(* Logix 5000 project; controller cal1615 1756-L62 rev 20.19; software revision 20.05; part 8 of 81 *)
(* tags used below, declared in another part *)
   AFI : BOOL;   // Always False Bit
   AutoT : PIDE_AUTOTUNE;
   FAULT : BOOL;   // Fault AFI
   HMI : BOOL;   // AFI HMI
   p01_dint_to_hmi : DINT[16];   // System Dint to HMI
   p01_param_heater_hl : REAL;   // Machine Parameter Heater HighTemperature Max Limit
   p01_param_process_air_hl : REAL;   // Machine Parameter Process Air High Limit
   p01_param_process_air_max : REAL;   // Machine Parameter Process Air High Temperature Max Setpoint Limit
   p01_param_temp_limit : REAL;   // Machine Parameter Maximum Temperature for Fan Operation
   p01_recipe_active : recipe;   // Active Recipe
   p01r01 : routine;
   p01r02 : routine;   // System Misc Control
   p01r02_all_fans_stopped : BOOL;   // System Misc Control All Fans Stopped
   p01r02_batch_run_time : DINT;   // System Misc Control Batch Minutes
   p01r02_batch_run_time_hrs : DINT;   // System Misc Control Batch Hours
   p01r02_ethernet_comm : DINT;
   p01r02_fault_exists : BOOL;
   p01r02_flash_bit : BOOL;   // System Misc Control Flash Bit
   p01r02_flash_timer_off : TIMER;   // System Misc Control Flash Timer Off
   p01r02_flash_timer_on : TIMER;   // System Misc Control Flash Timer On
   p01r02_plc_faults : DINT;   // System Misc Control PLC Faults
   p01r02_plc_scan_time : DINT;   // System PLC Scan Time
   p01r02_plc_scan_time_in_sec : REAL;   // System PLC Scan Time in Seconds
   p01r02_timer_batch : TIMER;   // System Misc Control Batch Timer Seconds
   p01r02_timer_fault : TIMER[25];   // System Misc Control Fault Dwell Timer
   p01r02_timer_half_second_off : TIMER;   // System Misc Control Timer Second Pulse Off
   p01r02_timer_half_second_on : TIMER;   // System Misc Control Timer 1/2 Second Pulse On
   p01r02_timer_second : TIMER[2];   // System Misc Control Timer Second Pulse
   p01r02_unack_fault : BOOL;   // System Misc Control Unacknowledged Fault Exists
   p01r02_unack_warning : BOOL;   // System Misc Control Unacknowledged Warning Exists
   p01r02_vfd_comm_2 : DINT[50];
   p01r02_warnings_exists : BOOL;
   p01r03 : routine;   // System Inputs
   p01r04 : routine;   // System Outputs
   p01r05 : routine;   // System Dint to HMI
   p01r06 : routine;   // System Real to HMI
   p01r07 : routine;   // System Alarms
   p01r08 : routine;   // System Warnings
   p01r09 : routine;   // System Modes
   p01r09_pb_global_reset : BOOL;   // System Modes PB: Global Fault Reset
   p01r10 : routine;   // System Annunciators
   p01r11 : routine;   // System Timer Presets
   p01r12 : routine;   // System Line Accel Decel Control
   p01r13 : routine;   // System Line Start Sequence
   p01r13_line_running : BOOL;   // System Line Start Sequence Line Running
   p02_dint_from_hmi : hmi_dint;
   p11r31_request_auto_run : BOOL;   // Zone 1 Exhaust Fan Run Request
   p11r32_request_auto_run : BOOL;   // Zone 1 Recirc Fan Run Request
   p12r31_request_auto_run : BOOL;   // Zone 2 Exhaust Fan Run Request
   p12r32_request_auto_run : BOOL;   // Zone 2 Recirc Fan Run Request
   p13r31_request_auto_run : BOOL;   // Zone 3 Exhaust Fan Run Request
   p13r32_request_auto_run : BOOL;   // Zone 3 Recirc Fan Run Request
   p23_do_enable_impreg_exhaust_fan : BOOL;   // Impreg Enclosure Digital Output Exhaust Fan Enable
   p23r13_request_auto_run : BOOL;   // Impreg Supply Fan VFD Request Auto Run
   p25_ai_ts2_lc : REAL;   // System Metering Roll VFD Minimum Start Tension
   p25r10_pid_manual_request : BOOL;
   p25r10_tension_request : BOOL;
   p25r20_pide_cv : REAL;

   p29r16_torque_acc_rate : REAL := 0.05;
   p29r16_torque_boost_acc_rate : REAL := 5000.0;
   p29r16_torque_boost_dec_rate : REAL := 2.0;
   p29r16_torque_boost_ref : REAL := 90.0;   // Winder Winder A VFD Request Jog REV
   p29r16_torque_boost_timer : TIMER := (PRE := 500);   // Zone 1 Exhaust VFD PB: Auto Stop
   p29r16_torque_dec_rate : REAL := 0.05;
   p29r16_torque_fast_acc_rate : REAL := 0.8;
   p29r16_torque_fast_dec_rate : REAL := 1.6;
   p29r16_torque_high_ref : REAL := 100.0;
   p29r16_torque_low_ref : REAL := 1.0;
   p29r16_torque_mode_acc_rate : REAL := 5000.0;
   p29r16_torque_mode_dec_rate : REAL := 4.0;
   p29r16_torque_ramp : SYS_ACC_DEC_RAMP := (IN_selected_line_speed := 100.0, IN_param_master_accel_rate := 0.05, IN_param_master_decel_rate := 0.05, IN_last_scan_s := 0.03255);
   p29r16_torque_soak_acc_rate : REAL := 0.05;
   p29r16_torque_soak_dec_rate : REAL := 0.05;
   p29r16_torque_start_timer : TIMER := (PRE := 200);   // Timer Winder B Torque Start Timer
   p29r16_vfd_start_request : BOOL := 1;
   p29r16_wdrb_accel_decel : SYS_ACC_DEC_RAMP := (IN_selected_line_speed := 16.283354, IN_param_master_accel_rate := 25.0, IN_param_master_decel_rate := 25.0, IN_last_scan_s := 0.03455);   // Winder Winder B VFD Accel Decel Ramp
   p29r16_wdrb_active : BOOL := 1;   // Winder Winder B VFD Active
   p29r16_wdrb_ramped_speed : REAL := 15.371705;   // Winder Winder B VFD Ramped Speed
   p29r16_zero_speed : BOOL;   // Winder Winder A VFD At Zero BSpeed
   p29r17 : routine := (comment := -1073741777);   // Winder Winder A Diameter
        .FAULT   // Winder Winder Turret VFD
        .UNACK_FAULT   // Winder Winder A Diameter Unacknowleged Faults Exist
        .UNACK_WARNING   // Winder Winder A Diameter Unacknowleged Warnings Exist
   p29r17_ave_control : CONTROL := (LEN := 19);   // Winder Winder A Diameter Calculation AVE Control
   p29r17_diameter_clac_active : BOOL;   // Winder Winder A Diameter Calculation Calc Active
   p29r17_selected_core_diameter : REAL := 3.25;   // Winder Winder A Diameter Calculation Selected Core Diameter
   p29r17_stack_ctrl : CONTROL := (LEN := 20, POS := 19);   // Winder Winder A Diameter Calculation Stack Control
   p29r17_timer : TIMER[5] := ([0].PRE := 20000, [1].PRE := 500);   // Winder Winder A Diameter Calculation Timers
        [1]   // Winder Winder A Diameter Calculation Sample Timer
   p29r17_timer_fault : TIMER[4];   // Winder Winder A Diameter Calculation Fault Dwell Timer
   p29r17_timer_warning : TIMER[4];   // Winder Winder A Diameter Calculation Warning Dwell Timer
   p29r17_web_speed_at_winder : REAL;   // Winder Winder A Diameter True Web Speed at the Winder Line Speed plus Accumulator Payout [fpm]
   p29r17_winder_a_actual_diam_inch : REAL := 6.327387;   // Winder Winder A Diameter Calculation Actual Diameter [in]
   p29r17_winder_a_avg_diam_inch : REAL := 6.2460294;   // Winder Winder A Diameter Calculation Winder A Average Diameter [in]
   p29r17_winder_a_calc_diam_inch : REAL := 6.327387;   // Winder Winder A Diameter Calculated Diameter Inch
   p29r17_winder_a_diam_avg_stack : REAL[1000] := ([0] := 6.227294, [1] := 6.2310367, [2] := 6.224801, [3] := 6.228541, [4] := 6.246055, [5] := 6.25359, [6] := 6.2360344, [7] := 6.2185774, [8] := 6.2148495, [9] := 6.216091, [10] := 6.247309, [11] := 6.2448, [12] := 6.2335353, [13] := 6.247309, [14] := 6.2737756, [15] := 6.277575, [16] := 6.304299, [17] := 6.3441668, [18] := 6.323527, [20] := 3.25, [21] := 3.25, [22] := 3.25, [23] := 3.25, [24] := 3.25, [25] := 3.25, [26] := 3.25, [27] := 3.25, [28] := 3.25, [29] := 3.25, [30] := 3.25, [31] := 3.25, [32] := 3.25, [33] := 3.25, [34] := 3.25, [35] := 3.25, [36] := 3.25, [37] := 3.25, [38] := 3.25, [39] := 3.25, [40] := 3.25, [41] := 3.25, [42] := 3.25, [43] := 3.25, [44] := 3.25, [45] := 3.25, [46] := 3.25, [47] := 3.25, [48] := 3.25, [49] := 3.25, [50] := 3.25, [51] := 3.25, [52] := 3.25, [53] := 3.25, [54] := 3.25, [55] := 3.25, [56] := 3.25, [57] := 3.25, [58] := 3.25, [59] := 3.25, [60] := 3.25,
        [61] := 3.25, [62] := 3.25, [63] := 3.25, [64] := 3.25, [65] := 3.25, [66] := 3.25, [67] := 3.25, [68] := 3.25, [69] := 3.25, [70] := 3.25, [71] := 3.25, [72] := 3.25, [73] := 3.25, [74] := 3.25, [75] := 3.25, [76] := 3.25, [77] := 3.25, [78] := 3.25, [79] := 3.25, [80] := 3.25, [81] := 3.25, [82] := 3.25, [83] := 3.25, [84] := 3.25, [85] := 3.25, [86] := 3.25, [87] := 3.25, [88] := 3.25, [89] := 3.25, [90] := 3.25, [91] := 3.25, [92] := 3.25, [93] := 3.25, [94] := 3.25, [95] := 3.25, [96] := 3.25, [97] := 3.25, [98] := 3.25, [99] := 3.25, [100] := 3.25, [101] := 3.25, [102] := 3.25, [103] := 3.25, [104] := 3.25, [105] := 3.25, [106] := 3.25, [107] := 3.25, [108] := 3.25, [109] := 3.25, [110] := 3.25, [111] := 3.25, [112] := 3.25, [113] := 3.25, [114] := 3.25, [115] := 3.25, [116] := 3.25, [117] := 3.25, [118] := 3.25, [119] := 3.25, [120] := 3.25,
        [121] := 3.25, [122] := 3.25, [123] := 3.25, [124] := 3.25, [125] := 3.25, [126] := 3.25, [127] := 3.25, [128] := 3.25, [129] := 3.25, [130] := 3.25, [131] := 3.25, [132] := 3.25, [133] := 3.25, [134] := 3.25, [135] := 3.25, [136] := 3.25, [137] := 3.25, [138] := 3.25, [139] := 3.25, [140] := 3.25, [141] := 3.25, [142] := 3.25, [143] := 3.25, [144] := 3.25, [145] := 3.25, [146] := 3.25, [147] := 3.25, [148] := 3.25, [149] := 3.25, [150] := 3.25, [151] := 3.25, [152] := 3.25, [153] := 3.25, [154] := 3.25, [155] := 3.25, [156] := 3.25, [157] := 3.25, [158] := 3.25, [159] := 3.25, [160] := 3.25, [161] := 3.25, [162] := 3.25, [163] := 3.25, [164] := 3.25, [165] := 3.25, [166] := 3.25, [167] := 3.25, [168] := 3.25, [169] := 3.25, [170] := 3.25, [171] := 3.25, [172] := 3.25, [173] := 3.25, [174] := 3.25, [175] := 3.25, [176] := 3.25, [177] := 3.25, [178] := 3.25, [179] := 3.25, [180] := 3.25,
        [181] := 3.25, [182] := 3.25, [183] := 3.25, [184] := 3.25, [185] := 3.25, [186] := 3.25, [187] := 3.25, [188] := 3.25, [189] := 3.25, [190] := 3.25, [191] := 3.25, [192] := 3.25, [193] := 3.25, [194] := 3.25, [195] := 3.25, [196] := 3.25, [197] := 3.25, [198] := 3.25, [199] := 3.25, [200] := 3.25, [201] := 3.25, [202] := 3.25, [203] := 3.25, [204] := 3.25, [205] := 3.25, [206] := 3.25, [207] := 3.25, [208] := 3.25, [209] := 3.25, [210] := 3.25, [211] := 3.25, [212] := 3.25, [213] := 3.25, [214] := 3.25, [215] := 3.25, [216] := 3.25, [217] := 3.25, [218] := 3.25, [219] := 3.25, [220] := 3.25, [221] := 3.25, [222] := 3.25, [223] := 3.25, [224] := 3.25, [225] := 3.25, [226] := 3.25, [227] := 3.25, [228] := 3.25, [229] := 3.25, [230] := 3.25, [231] := 3.25, [232] := 3.25, [233] := 3.25, [234] := 3.25, [235] := 3.25, [236] := 3.25, [237] := 3.25, [238] := 3.25, [239] := 3.25, [240] := 3.25,
        [241] := 3.25, [242] := 3.25, [243] := 3.25, [244] := 3.25, [245] := 3.25, [246] := 3.25, [247] := 3.25, [248] := 3.25, [249] := 3.25, [250] := 3.25, [251] := 3.25, [252] := 3.25, [253] := 3.25, [254] := 3.25, [255] := 3.25, [256] := 3.25, [257] := 3.25, [258] := 3.25, [259] := 3.25, [260] := 3.25, [261] := 3.25, [262] := 3.25, [263] := 3.25, [264] := 3.25, [265] := 3.25, [266] := 3.25, [267] := 3.25, [268] := 3.25, [269] := 3.25, [270] := 3.25, [271] := 3.25, [272] := 3.25, [273] := 3.25, [274] := 3.25, [275] := 3.25, [276] := 3.25, [277] := 3.25, [278] := 3.25, [279] := 3.25, [280] := 3.25, [281] := 3.25, [282] := 3.25, [283] := 3.25, [284] := 3.25, [285] := 3.25, [286] := 3.25, [287] := 3.25, [288] := 3.25, [289] := 3.25, [290] := 3.25, [291] := 3.25, [292] := 3.25, [293] := 3.25, [294] := 3.25, [295] := 3.25, [296] := 3.25, [297] := 3.25, [298] := 3.25, [299] := 3.25, [300] := 3.25,
        [301] := 3.25, [302] := 3.25, [303] := 3.25, [304] := 3.25, [305] := 3.25, [306] := 3.25, [307] := 3.25, [308] := 3.25, [309] := 3.25, [310] := 3.25, [311] := 3.25, [312] := 3.25, [313] := 3.25, [314] := 3.25, [315] := 3.25, [316] := 3.25, [317] := 3.25, [318] := 3.25, [319] := 3.25, [320] := 3.25, [321] := 3.25, [322] := 3.25, [323] := 3.25, [324] := 3.25, [325] := 3.25, [326] := 3.25, [327] := 3.25, [328] := 3.25, [329] := 3.25, [330] := 3.25, [331] := 3.25, [332] := 3.25, [333] := 3.25, [334] := 3.25, [335] := 3.25, [336] := 3.25, [337] := 3.25, [338] := 3.25, [339] := 3.25, [340] := 3.25, [341] := 3.25, [342] := 3.25, [343] := 3.25, [344] := 3.25, [345] := 3.25, [346] := 3.25, [347] := 3.25, [348] := 3.25, [349] := 3.25, [350] := 3.25, [351] := 3.25, [352] := 3.25, [353] := 3.25, [354] := 3.25, [355] := 3.25, [356] := 3.25, [357] := 3.25, [358] := 3.25, [359] := 3.25, [360] := 3.25,
        [361] := 3.25, [362] := 3.25, [363] := 3.25, [364] := 3.25, [365] := 3.25, [366] := 3.25, [367] := 3.25, [368] := 3.25, [369] := 3.25, [370] := 3.25, [371] := 3.25, [372] := 3.25, [373] := 3.25, [374] := 3.25, [375] := 3.25, [376] := 3.25, [377] := 3.25, [378] := 3.25, [379] := 3.25, [380] := 3.25, [381] := 3.25, [382] := 3.25, [383] := 3.25, [384] := 3.25, [385] := 3.25, [386] := 3.25, [387] := 3.25, [388] := 3.25, [389] := 3.25, [390] := 3.25, [391] := 3.25, [392] := 3.25, [393] := 3.25, [394] := 3.25, [395] := 3.25, [396] := 3.25, [397] := 3.25, [398] := 3.25, [399] := 3.25, [400] := 3.25, [401] := 3.25, [402] := 3.25, [403] := 3.25, [404] := 3.25, [405] := 3.25, [406] := 3.25, [407] := 3.25, [408] := 3.25, [409] := 3.25, [410] := 3.25, [411] := 3.25, [412] := 3.25, [413] := 3.25, [414] := 3.25, [415] := 3.25, [416] := 3.25, [417] := 3.25, [418] := 3.25, [419] := 3.25, [420] := 3.25,
        [421] := 3.25, [422] := 3.25, [423] := 3.25, [424] := 3.25, [425] := 3.25, [426] := 3.25, [427] := 3.25, [428] := 3.25, [429] := 3.25, [430] := 3.25, [431] := 3.25, [432] := 3.25, [433] := 3.25, [434] := 3.25, [435] := 3.25, [436] := 3.25, [437] := 3.25, [438] := 3.25, [439] := 3.25, [440] := 3.25, [441] := 3.25, [442] := 3.25, [443] := 3.25, [444] := 3.25, [445] := 3.25, [446] := 3.25, [447] := 3.25, [448] := 3.25, [449] := 3.25, [450] := 3.25, [451] := 3.25, [452] := 3.25, [453] := 3.25, [454] := 3.25, [455] := 3.25, [456] := 3.25, [457] := 3.25, [458] := 3.25, [459] := 3.25, [460] := 3.25, [461] := 3.25, [462] := 3.25, [463] := 3.25, [464] := 3.25, [465] := 3.25, [466] := 3.25, [467] := 3.25, [468] := 3.25, [469] := 3.25, [470] := 3.25, [471] := 3.25, [472] := 3.25, [473] := 3.25, [474] := 3.25, [475] := 3.25, [476] := 3.25, [477] := 3.25, [478] := 3.25, [479] := 3.25, [480] := 3.25,
        [481] := 3.25, [482] := 3.25, [483] := 3.25, [484] := 3.25, [485] := 3.25, [486] := 3.25, [487] := 3.25, [488] := 3.25, [489] := 3.25, [490] := 3.25, [491] := 3.25, [492] := 3.25, [493] := 3.25, [494] := 3.25, [495] := 3.25, [496] := 3.25, [497] := 3.25, [498] := 3.25, [499] := 3.25, [500] := 3.25, [501] := 3.25, [502] := 3.25, [503] := 3.25, [504] := 3.25, [505] := 3.25, [506] := 3.25, [507] := 3.25, [508] := 3.25, [509] := 3.25, [510] := 3.25, [511] := 3.25, [512] := 3.25, [513] := 3.25, [514] := 3.25, [515] := 3.25, [516] := 3.25, [517] := 3.25, [518] := 3.25, [519] := 3.25, [520] := 3.25, [521] := 3.25, [522] := 3.25, [523] := 3.25, [524] := 3.25, [525] := 3.25, [526] := 3.25, [527] := 3.25, [528] := 3.25, [529] := 3.25, [530] := 3.25, [531] := 3.25, [532] := 3.25, [533] := 3.25, [534] := 3.25, [535] := 3.25, [536] := 3.25, [537] := 3.25, [538] := 3.25, [539] := 3.25, [540] := 3.25,
        [541] := 3.25, [542] := 3.25, [543] := 3.25, [544] := 3.25, [545] := 3.25, [546] := 3.25, [547] := 3.25, [548] := 3.25, [549] := 3.25, [550] := 3.25, [551] := 3.25, [552] := 3.25, [553] := 3.25, [554] := 3.25, [555] := 3.25, [556] := 3.25, [557] := 3.25, [558] := 3.25, [559] := 3.25, [560] := 3.25, [561] := 3.25, [562] := 3.25, [563] := 3.25, [564] := 3.25, [565] := 3.25, [566] := 3.25, [567] := 3.25, [568] := 3.25, [569] := 3.25, [570] := 3.25, [571] := 3.25, [572] := 3.25, [573] := 3.25, [574] := 3.25, [575] := 3.25, [576] := 3.25, [577] := 3.25, [578] := 3.25, [579] := 3.25, [580] := 3.25, [581] := 3.25, [582] := 3.25, [583] := 3.25, [584] := 3.25, [585] := 3.25, [586] := 3.25, [587] := 3.25, [588] := 3.25, [589] := 3.25, [590] := 3.25, [591] := 3.25, [592] := 3.25, [593] := 3.25, [594] := 3.25, [595] := 3.25, [596] := 3.25, [597] := 3.25, [598] := 3.25, [599] := 3.25, [600] := 3.25,
        [601] := 3.25, [602] := 3.25, [603] := 3.25, [604] := 3.25, [605] := 3.25, [606] := 3.25, [607] := 3.25, [608] := 3.25, [609] := 3.25, [610] := 3.25, [611] := 3.25, [612] := 3.25, [613] := 3.25, [614] := 3.25, [615] := 3.25, [616] := 3.25, [617] := 3.25, [618] := 3.25, [619] := 3.25, [620] := 3.25, [621] := 3.25, [622] := 3.25, [623] := 3.25, [624] := 3.25, [625] := 3.25, [626] := 3.25, [627] := 3.25, [628] := 3.25, [629] := 3.25, [630] := 3.25, [631] := 3.25, [632] := 3.25, [633] := 3.25, [634] := 3.25, [635] := 3.25, [636] := 3.25, [637] := 3.25, [638] := 3.25, [639] := 3.25, [640] := 3.25, [641] := 3.25, [642] := 3.25, [643] := 3.25, [644] := 3.25, [645] := 3.25, [646] := 3.25, [647] := 3.25, [648] := 3.25, [649] := 3.25, [650] := 3.25, [651] := 3.25, [652] := 3.25, [653] := 3.25, [654] := 3.25, [655] := 3.25, [656] := 3.25, [657] := 3.25, [658] := 3.25, [659] := 3.25, [660] := 3.25,
        [661] := 3.25, [662] := 3.25, [663] := 3.25, [664] := 3.25, [665] := 3.25, [666] := 3.25, [667] := 3.25, [668] := 3.25, [669] := 3.25, [670] := 3.25, [671] := 3.25, [672] := 3.25, [673] := 3.25, [674] := 3.25, [675] := 3.25, [676] := 3.25, [677] := 3.25, [678] := 3.25, [679] := 3.25, [680] := 3.25, [681] := 3.25, [682] := 3.25, [683] := 3.25, [684] := 3.25, [685] := 3.25, [686] := 3.25, [687] := 3.25, [688] := 3.25, [689] := 3.25, [690] := 3.25, [691] := 3.25, [692] := 3.25, [693] := 3.25, [694] := 3.25, [695] := 3.25, [696] := 3.25, [697] := 3.25, [698] := 3.25, [699] := 3.25, [700] := 3.25, [701] := 3.25, [702] := 3.25, [703] := 3.25, [704] := 3.25, [705] := 3.25, [706] := 3.25, [707] := 3.25, [708] := 3.25, [709] := 3.25, [710] := 3.25, [711] := 3.25, [712] := 3.25, [713] := 3.25, [714] := 3.25, [715] := 3.25, [716] := 3.25, [717] := 3.25, [718] := 3.25, [719] := 3.25, [720] := 3.25,
        [721] := 3.25, [722] := 3.25, [723] := 3.25, [724] := 3.25, [725] := 3.25, [726] := 3.25, [727] := 3.25, [728] := 3.25, [729] := 3.25, [730] := 3.25, [731] := 3.25, [732] := 3.25, [733] := 3.25, [734] := 3.25, [735] := 3.25, [736] := 3.25, [737] := 3.25, [738] := 3.25, [739] := 3.25, [740] := 3.25, [741] := 3.25, [742] := 3.25, [743] := 3.25, [744] := 3.25, [745] := 3.25, [746] := 3.25, [747] := 3.25, [748] := 3.25, [749] := 3.25, [750] := 3.25, [751] := 3.25, [752] := 3.25, [753] := 3.25, [754] := 3.25, [755] := 3.25, [756] := 3.25, [757] := 3.25, [758] := 3.25, [759] := 3.25, [760] := 3.25, [761] := 3.25, [762] := 3.25, [763] := 3.25, [764] := 3.25, [765] := 3.25, [766] := 3.25, [767] := 3.25, [768] := 3.25, [769] := 3.25, [770] := 3.25, [771] := 3.25, [772] := 3.25, [773] := 3.25, [774] := 3.25, [775] := 3.25, [776] := 3.25, [777] := 3.25, [778] := 3.25, [779] := 3.25, [780] := 3.25,
        [781] := 3.25, [782] := 3.25, [783] := 3.25, [784] := 3.25, [785] := 3.25, [786] := 3.25, [787] := 3.25, [788] := 3.25, [789] := 3.25, [790] := 3.25, [791] := 3.25, [792] := 3.25, [793] := 3.25, [794] := 3.25, [795] := 3.25, [796] := 3.25, [797] := 3.25, [798] := 3.25, [799] := 3.25, [800] := 3.25, [801] := 3.25, [802] := 3.25, [803] := 3.25, [804] := 3.25, [805] := 3.25, [806] := 3.25, [807] := 3.25, [808] := 3.25, [809] := 3.25, [810] := 3.25, [811] := 3.25, [812] := 3.25, [813] := 3.25, [814] := 3.25, [815] := 3.25, [816] := 3.25, [817] := 3.25, [818] := 3.25, [819] := 3.25, [820] := 3.25, [821] := 3.25, [822] := 3.25, [823] := 3.25, [824] := 3.25, [825] := 3.25, [826] := 3.25, [827] := 3.25, [828] := 3.25, [829] := 3.25, [830] := 3.25, [831] := 3.25, [832] := 3.25, [833] := 3.25, [834] := 3.25, [835] := 3.25, [836] := 3.25, [837] := 3.25, [838] := 3.25, [839] := 3.25, [840] := 3.25,
        [841] := 3.25, [842] := 3.25, [843] := 3.25, [844] := 3.25, [845] := 3.25, [846] := 3.25, [847] := 3.25, [848] := 3.25, [849] := 3.25, [850] := 3.25, [851] := 3.25, [852] := 3.25, [853] := 3.25, [854] := 3.25, [855] := 3.25, [856] := 3.25, [857] := 3.25, [858] := 3.25, [859] := 3.25, [860] := 3.25, [861] := 3.25, [862] := 3.25, [863] := 3.25, [864] := 3.25, [865] := 3.25, [866] := 3.25, [867] := 3.25, [868] := 3.25, [869] := 3.25, [870] := 3.25, [871] := 3.25, [872] := 3.25, [873] := 3.25, [874] := 3.25, [875] := 3.25, [876] := 3.25, [877] := 3.25, [878] := 3.25, [879] := 3.25, [880] := 3.25, [881] := 3.25, [882] := 3.25, [883] := 3.25, [884] := 3.25, [885] := 3.25, [886] := 3.25, [887] := 3.25, [888] := 3.25, [889] := 3.25, [890] := 3.25, [891] := 3.25, [892] := 3.25, [893] := 3.25, [894] := 3.25, [895] := 3.25, [896] := 3.25, [897] := 3.25, [898] := 3.25, [899] := 3.25, [900] := 3.25,
        [901] := 3.25, [902] := 3.25, [903] := 3.25, [904] := 3.25, [905] := 3.25, [906] := 3.25, [907] := 3.25, [908] := 3.25, [909] := 3.25, [910] := 3.25, [911] := 3.25, [912] := 3.25, [913] := 3.25, [914] := 3.25, [915] := 3.25, [916] := 3.25, [917] := 3.25, [918] := 3.25, [919] := 3.25, [920] := 3.25, [921] := 3.25, [922] := 3.25, [923] := 3.25, [924] := 3.25, [925] := 3.25, [926] := 3.25, [927] := 3.25, [928] := 3.25, [929] := 3.25, [930] := 3.25, [931] := 3.25, [932] := 3.25, [933] := 3.25, [934] := 3.25, [935] := 3.25, [936] := 3.25, [937] := 3.25, [938] := 3.25, [939] := 3.25, [940] := 3.25, [941] := 3.25, [942] := 3.25, [943] := 3.25, [944] := 3.25, [945] := 3.25, [946] := 3.25, [947] := 3.25, [948] := 3.25, [949] := 3.25, [950] := 3.25, [951] := 3.25, [952] := 3.25, [953] := 3.25, [954] := 3.25, [955] := 3.25, [956] := 3.25, [957] := 3.25, [958] := 3.25, [959] := 3.25, [960] := 3.25,
        [961] := 3.25, [962] := 3.25, [963] := 3.25, [964] := 3.25, [965] := 3.25, [966] := 3.25, [967] := 3.25, [968] := 3.25, [969] := 3.25, [970] := 3.25, [971] := 3.25, [972] := 3.25, [973] := 3.25, [974] := 3.25, [975] := 3.25, [976] := 3.25, [977] := 3.25, [978] := 3.25, [979] := 3.25, [980] := 3.25, [981] := 3.25, [982] := 3.25, [983] := 3.25, [984] := 3.25, [985] := 3.25, [986] := 3.25, [987] := 3.25, [988] := 3.25, [989] := 3.25, [990] := 3.25, [991] := 3.25, [992] := 3.25, [993] := 3.25, [994] := 3.25, [995] := 3.25, [996] := 3.25, [997] := 3.25, [998] := 3.25, [999] := 3.25);
   p29r17_winder_a_selected_diam_inch : REAL := 3.25;   // Winder Winder A Diameter Calculation Winder Selected Diameter [in]
   p29r17_winder_a_unload : REAL := 6.2049294;
   p29r18 : routine := (comment := -1073741777);   // Winder Winder B Diameter
        .UNACK_FAULT   // Winder Winder B Diameter Unacknowleged Faults Exist
        .UNACK_WARNING   // Winder Winder B Diameter Unacknowleged Warnings Exist
   p29r18_ave_control : CONTROL := (LEN := 19);   // Winder Winder A Diameter Calculation AVE Control
   p29r18_diameter_calc_active : BOOL := 1;   // Winder Winder B Diameter Calculation Calculation Active
   p29r18_min_tension : REAL := 10.0;   // Winder Winder B Diameter Calc Minimum Tension
   p29r18_selected_core_diameter : REAL := 3.25;   // Winder Winder B Diameter Calculation Selected Core Diameter
   p29r18_stack_ctrl : CONTROL := (LEN := 20, POS := 20, EN := 1, DN := 1);   // Winder Winder B Diameter Calculation FiFo Control
   p29r18_timer : TIMER[5] := ([0].PRE := 20000, [0].ACC := 20017, [0].EN := 1, [0].DN := 1, [1].PRE := 500, [1].ACC := 466, [1].EN := 1, [1].TT := 1);   // Winder Winder B Diameter Calculation Timers
   p29r18_timer_fault : TIMER[4];   // Winder Winder B Diameter Calculation Fault Dwell Timer
   p29r18_timer_warning : TIMER[4];   // Winder Winder B Diameter Warning Dwell Timer
   p29r18_web_speed_at_winder : REAL;   // Winder Winder B Diameter True Web Speed at the Winder Line Speed plus Accumulator Payout [fpm]
   p29r18_winder_b_actual_diam_inch : REAL := 7.2323503;   // Winder Winder B Diameter Calculation Actual Diameter [in]
   p29r18_winder_b_avg_diam_inch : REAL := 6.935298;   // Winder Winder B Diameter Calculation Average Diameter [in]
   p29r18_winder_b_calc_diam_inch : REAL := 7.21557;   // Winder Winder B Diameter Calculated Diameter Inch
   p29r18_winder_b_diam_avg_stack : REAL[1000] := ([0] := 7.30026, [1] := 7.30026, [2] := 7.30026, [3] := 7.30026, [4] := 7.30026, [5] := 7.30026, [6] := 7.21557, [7] := 7.2323503, [8] := 7.266146, [9] := 7.283163, [10] := 7.266146, [11] := 7.249209, [12] := 7.249209, [13] := 7.21557, [14] := 7.1988673, [15] := 7.1988673, [16] := 7.2323503, [17] := 7.283163, [18] := 7.30026, [20] := 3.25, [21] := 3.25, [22] := 3.25, [23] := 3.25, [24] := 3.25, [25] := 3.25, [26] := 3.25, [27] := 3.25, [28] := 3.25, [29] := 3.25, [30] := 3.25, [31] := 3.25, [32] := 3.25, [33] := 3.25, [34] := 3.25, [35] := 3.25, [36] := 3.25, [37] := 3.25, [38] := 3.25, [39] := 3.25, [40] := 3.25, [41] := 3.25, [42] := 3.25, [43] := 3.25, [44] := 3.25, [45] := 3.25, [46] := 3.25, [47] := 3.25, [48] := 3.25, [49] := 3.25, [50] := 3.25, [51] := 3.25, [52] := 3.25, [53] := 3.25, [54] := 3.25, [55] := 3.25, [56] := 3.25, [57] := 3.25, [58] := 3.25, [59] := 3.25, [60] := 3.25,
        [61] := 3.25, [62] := 3.25, [63] := 3.25, [64] := 3.25, [65] := 3.25, [66] := 3.25, [67] := 3.25, [68] := 3.25, [69] := 3.25, [70] := 3.25, [71] := 3.25, [72] := 3.25, [73] := 3.25, [74] := 3.25, [75] := 3.25, [76] := 3.25, [77] := 3.25, [78] := 3.25, [79] := 3.25, [80] := 3.25, [81] := 3.25, [82] := 3.25, [83] := 3.25, [84] := 3.25, [85] := 3.25, [86] := 3.25, [87] := 3.25, [88] := 3.25, [89] := 3.25, [90] := 3.25, [91] := 3.25, [92] := 3.25, [93] := 3.25, [94] := 3.25, [95] := 3.25, [96] := 3.25, [97] := 3.25, [98] := 3.25, [99] := 3.25, [100] := 3.25, [101] := 3.25, [102] := 3.25, [103] := 3.25, [104] := 3.25, [105] := 3.25, [106] := 3.25, [107] := 3.25, [108] := 3.25, [109] := 3.25, [110] := 3.25, [111] := 3.25, [112] := 3.25, [113] := 3.25, [114] := 3.25, [115] := 3.25, [116] := 3.25, [117] := 3.25, [118] := 3.25, [119] := 3.25, [120] := 3.25,
        [121] := 3.25, [122] := 3.25, [123] := 3.25, [124] := 3.25, [125] := 3.25, [126] := 3.25, [127] := 3.25, [128] := 3.25, [129] := 3.25, [130] := 3.25, [131] := 3.25, [132] := 3.25, [133] := 3.25, [134] := 3.25, [135] := 3.25, [136] := 3.25, [137] := 3.25, [138] := 3.25, [139] := 3.25, [140] := 3.25, [141] := 3.25, [142] := 3.25, [143] := 3.25, [144] := 3.25, [145] := 3.25, [146] := 3.25, [147] := 3.25, [148] := 3.25, [149] := 3.25, [150] := 3.25, [151] := 3.25, [152] := 3.25, [153] := 3.25, [154] := 3.25, [155] := 3.25, [156] := 3.25, [157] := 3.25, [158] := 3.25, [159] := 3.25, [160] := 3.25, [161] := 3.25, [162] := 3.25, [163] := 3.25, [164] := 3.25, [165] := 3.25, [166] := 3.25, [167] := 3.25, [168] := 3.25, [169] := 3.25, [170] := 3.25, [171] := 3.25, [172] := 3.25, [173] := 3.25, [174] := 3.25, [175] := 3.25, [176] := 3.25, [177] := 3.25, [178] := 3.25, [179] := 3.25, [180] := 3.25,
        [181] := 3.25, [182] := 3.25, [183] := 3.25, [184] := 3.25, [185] := 3.25, [186] := 3.25, [187] := 3.25, [188] := 3.25, [189] := 3.25, [190] := 3.25, [191] := 3.25, [192] := 3.25, [193] := 3.25, [194] := 3.25, [195] := 3.25, [196] := 3.25, [197] := 3.25, [198] := 3.25, [199] := 3.25, [200] := 3.25, [201] := 3.25, [202] := 3.25, [203] := 3.25, [204] := 3.25, [205] := 3.25, [206] := 3.25, [207] := 3.25, [208] := 3.25, [209] := 3.25, [210] := 3.25, [211] := 3.25, [212] := 3.25, [213] := 3.25, [214] := 3.25, [215] := 3.25, [216] := 3.25, [217] := 3.25, [218] := 3.25, [219] := 3.25, [220] := 3.25, [221] := 3.25, [222] := 3.25, [223] := 3.25, [224] := 3.25, [225] := 3.25, [226] := 3.25, [227] := 3.25, [228] := 3.25, [229] := 3.25, [230] := 3.25, [231] := 3.25, [232] := 3.25, [233] := 3.25, [234] := 3.25, [235] := 3.25, [236] := 3.25, [237] := 3.25, [238] := 3.25, [239] := 3.25, [240] := 3.25,
        [241] := 3.25, [242] := 3.25, [243] := 3.25, [244] := 3.25, [245] := 3.25, [246] := 3.25, [247] := 3.25, [248] := 3.25, [249] := 3.25, [250] := 3.25, [251] := 3.25, [252] := 3.25, [253] := 3.25, [254] := 3.25, [255] := 3.25, [256] := 3.25, [257] := 3.25, [258] := 3.25, [259] := 3.25, [260] := 3.25, [261] := 3.25, [262] := 3.25, [263] := 3.25, [264] := 3.25, [265] := 3.25, [266] := 3.25, [267] := 3.25, [268] := 3.25, [269] := 3.25, [270] := 3.25, [271] := 3.25, [272] := 3.25, [273] := 3.25, [274] := 3.25, [275] := 3.25, [276] := 3.25, [277] := 3.25, [278] := 3.25, [279] := 3.25, [280] := 3.25, [281] := 3.25, [282] := 3.25, [283] := 3.25, [284] := 3.25, [285] := 3.25, [286] := 3.25, [287] := 3.25, [288] := 3.25, [289] := 3.25, [290] := 3.25, [291] := 3.25, [292] := 3.25, [293] := 3.25, [294] := 3.25, [295] := 3.25, [296] := 3.25, [297] := 3.25, [298] := 3.25, [299] := 3.25, [300] := 3.25,
        [301] := 3.25, [302] := 3.25, [303] := 3.25, [304] := 3.25, [305] := 3.25, [306] := 3.25, [307] := 3.25, [308] := 3.25, [309] := 3.25, [310] := 3.25, [311] := 3.25, [312] := 3.25, [313] := 3.25, [314] := 3.25, [315] := 3.25, [316] := 3.25, [317] := 3.25, [318] := 3.25, [319] := 3.25, [320] := 3.25, [321] := 3.25, [322] := 3.25, [323] := 3.25, [324] := 3.25, [325] := 3.25, [326] := 3.25, [327] := 3.25, [328] := 3.25, [329] := 3.25, [330] := 3.25, [331] := 3.25, [332] := 3.25, [333] := 3.25, [334] := 3.25, [335] := 3.25, [336] := 3.25, [337] := 3.25, [338] := 3.25, [339] := 3.25, [340] := 3.25, [341] := 3.25, [342] := 3.25, [343] := 3.25, [344] := 3.25, [345] := 3.25, [346] := 3.25, [347] := 3.25, [348] := 3.25, [349] := 3.25, [350] := 3.25, [351] := 3.25, [352] := 3.25, [353] := 3.25, [354] := 3.25, [355] := 3.25, [356] := 3.25, [357] := 3.25, [358] := 3.25, [359] := 3.25, [360] := 3.25,
        [361] := 3.25, [362] := 3.25, [363] := 3.25, [364] := 3.25, [365] := 3.25, [366] := 3.25, [367] := 3.25, [368] := 3.25, [369] := 3.25, [370] := 3.25, [371] := 3.25, [372] := 3.25, [373] := 3.25, [374] := 3.25, [375] := 3.25, [376] := 3.25, [377] := 3.25, [378] := 3.25, [379] := 3.25, [380] := 3.25, [381] := 3.25, [382] := 3.25, [383] := 3.25, [384] := 3.25, [385] := 3.25, [386] := 3.25, [387] := 3.25, [388] := 3.25, [389] := 3.25, [390] := 3.25, [391] := 3.25, [392] := 3.25, [393] := 3.25, [394] := 3.25, [395] := 3.25, [396] := 3.25, [397] := 3.25, [398] := 3.25, [399] := 3.25, [400] := 3.25, [401] := 3.25, [402] := 3.25, [403] := 3.25, [404] := 3.25, [405] := 3.25, [406] := 3.25, [407] := 3.25, [408] := 3.25, [409] := 3.25, [410] := 3.25, [411] := 3.25, [412] := 3.25, [413] := 3.25, [414] := 3.25, [415] := 3.25, [416] := 3.25, [417] := 3.25, [418] := 3.25, [419] := 3.25, [420] := 3.25,
        [421] := 3.25, [422] := 3.25, [423] := 3.25, [424] := 3.25, [425] := 3.25, [426] := 3.25, [427] := 3.25, [428] := 3.25, [429] := 3.25, [430] := 3.25, [431] := 3.25, [432] := 3.25, [433] := 3.25, [434] := 3.25, [435] := 3.25, [436] := 3.25, [437] := 3.25, [438] := 3.25, [439] := 3.25, [440] := 3.25, [441] := 3.25, [442] := 3.25, [443] := 3.25, [444] := 3.25, [445] := 3.25, [446] := 3.25, [447] := 3.25, [448] := 3.25, [449] := 3.25, [450] := 3.25, [451] := 3.25, [452] := 3.25, [453] := 3.25, [454] := 3.25, [455] := 3.25, [456] := 3.25, [457] := 3.25, [458] := 3.25, [459] := 3.25, [460] := 3.25, [461] := 3.25, [462] := 3.25, [463] := 3.25, [464] := 3.25, [465] := 3.25, [466] := 3.25, [467] := 3.25, [468] := 3.25, [469] := 3.25, [470] := 3.25, [471] := 3.25, [472] := 3.25, [473] := 3.25, [474] := 3.25, [475] := 3.25, [476] := 3.25, [477] := 3.25, [478] := 3.25, [479] := 3.25, [480] := 3.25,
        [481] := 3.25, [482] := 3.25, [483] := 3.25, [484] := 3.25, [485] := 3.25, [486] := 3.25, [487] := 3.25, [488] := 3.25, [489] := 3.25, [490] := 3.25, [491] := 3.25, [492] := 3.25, [493] := 3.25, [494] := 3.25, [495] := 3.25, [496] := 3.25, [497] := 3.25, [498] := 3.25, [499] := 3.25, [500] := 3.25, [501] := 3.25, [502] := 3.25, [503] := 3.25, [504] := 3.25, [505] := 3.25, [506] := 3.25, [507] := 3.25, [508] := 3.25, [509] := 3.25, [510] := 3.25, [511] := 3.25, [512] := 3.25, [513] := 3.25, [514] := 3.25, [515] := 3.25, [516] := 3.25, [517] := 3.25, [518] := 3.25, [519] := 3.25, [520] := 3.25, [521] := 3.25, [522] := 3.25, [523] := 3.25, [524] := 3.25, [525] := 3.25, [526] := 3.25, [527] := 3.25, [528] := 3.25, [529] := 3.25, [530] := 3.25, [531] := 3.25, [532] := 3.25, [533] := 3.25, [534] := 3.25, [535] := 3.25, [536] := 3.25, [537] := 3.25, [538] := 3.25, [539] := 3.25, [540] := 3.25,
        [541] := 3.25, [542] := 3.25, [543] := 3.25, [544] := 3.25, [545] := 3.25, [546] := 3.25, [547] := 3.25, [548] := 3.25, [549] := 3.25, [550] := 3.25, [551] := 3.25, [552] := 3.25, [553] := 3.25, [554] := 3.25, [555] := 3.25, [556] := 3.25, [557] := 3.25, [558] := 3.25, [559] := 3.25, [560] := 3.25, [561] := 3.25, [562] := 3.25, [563] := 3.25, [564] := 3.25, [565] := 3.25, [566] := 3.25, [567] := 3.25, [568] := 3.25, [569] := 3.25, [570] := 3.25, [571] := 3.25, [572] := 3.25, [573] := 3.25, [574] := 3.25, [575] := 3.25, [576] := 3.25, [577] := 3.25, [578] := 3.25, [579] := 3.25, [580] := 3.25, [581] := 3.25, [582] := 3.25, [583] := 3.25, [584] := 3.25, [585] := 3.25, [586] := 3.25, [587] := 3.25, [588] := 3.25, [589] := 3.25, [590] := 3.25, [591] := 3.25, [592] := 3.25, [593] := 3.25, [594] := 3.25, [595] := 3.25, [596] := 3.25, [597] := 3.25, [598] := 3.25, [599] := 3.25, [600] := 3.25,
        [601] := 3.25, [602] := 3.25, [603] := 3.25, [604] := 3.25, [605] := 3.25, [606] := 3.25, [607] := 3.25, [608] := 3.25, [609] := 3.25, [610] := 3.25, [611] := 3.25, [612] := 3.25, [613] := 3.25, [614] := 3.25, [615] := 3.25, [616] := 3.25, [617] := 3.25, [618] := 3.25, [619] := 3.25, [620] := 3.25, [621] := 3.25, [622] := 3.25, [623] := 3.25, [624] := 3.25, [625] := 3.25, [626] := 3.25, [627] := 3.25, [628] := 3.25, [629] := 3.25, [630] := 3.25, [631] := 3.25, [632] := 3.25, [633] := 3.25, [634] := 3.25, [635] := 3.25, [636] := 3.25, [637] := 3.25, [638] := 3.25, [639] := 3.25, [640] := 3.25, [641] := 3.25, [642] := 3.25, [643] := 3.25, [644] := 3.25, [645] := 3.25, [646] := 3.25, [647] := 3.25, [648] := 3.25, [649] := 3.25, [650] := 3.25, [651] := 3.25, [652] := 3.25, [653] := 3.25, [654] := 3.25, [655] := 3.25, [656] := 3.25, [657] := 3.25, [658] := 3.25, [659] := 3.25, [660] := 3.25,
        [661] := 3.25, [662] := 3.25, [663] := 3.25, [664] := 3.25, [665] := 3.25, [666] := 3.25, [667] := 3.25, [668] := 3.25, [669] := 3.25, [670] := 3.25, [671] := 3.25, [672] := 3.25, [673] := 3.25, [674] := 3.25, [675] := 3.25, [676] := 3.25, [677] := 3.25, [678] := 3.25, [679] := 3.25, [680] := 3.25, [681] := 3.25, [682] := 3.25, [683] := 3.25, [684] := 3.25, [685] := 3.25, [686] := 3.25, [687] := 3.25, [688] := 3.25, [689] := 3.25, [690] := 3.25, [691] := 3.25, [692] := 3.25, [693] := 3.25, [694] := 3.25, [695] := 3.25, [696] := 3.25, [697] := 3.25, [698] := 3.25, [699] := 3.25, [700] := 3.25, [701] := 3.25, [702] := 3.25, [703] := 3.25, [704] := 3.25, [705] := 3.25, [706] := 3.25, [707] := 3.25, [708] := 3.25, [709] := 3.25, [710] := 3.25, [711] := 3.25, [712] := 3.25, [713] := 3.25, [714] := 3.25, [715] := 3.25, [716] := 3.25, [717] := 3.25, [718] := 3.25, [719] := 3.25, [720] := 3.25,
        [721] := 3.25, [722] := 3.25, [723] := 3.25, [724] := 3.25, [725] := 3.25, [726] := 3.25, [727] := 3.25, [728] := 3.25, [729] := 3.25, [730] := 3.25, [731] := 3.25, [732] := 3.25, [733] := 3.25, [734] := 3.25, [735] := 3.25, [736] := 3.25, [737] := 3.25, [738] := 3.25, [739] := 3.25, [740] := 3.25, [741] := 3.25, [742] := 3.25, [743] := 3.25, [744] := 3.25, [745] := 3.25, [746] := 3.25, [747] := 3.25, [748] := 3.25, [749] := 3.25, [750] := 3.25, [751] := 3.25, [752] := 3.25, [753] := 3.25, [754] := 3.25, [755] := 3.25, [756] := 3.25, [757] := 3.25, [758] := 3.25, [759] := 3.25, [760] := 3.25, [761] := 3.25, [762] := 3.25, [763] := 3.25, [764] := 3.25, [765] := 3.25, [766] := 3.25, [767] := 3.25, [768] := 3.25, [769] := 3.25, [770] := 3.25, [771] := 3.25, [772] := 3.25, [773] := 3.25, [774] := 3.25, [775] := 3.25, [776] := 3.25, [777] := 3.25, [778] := 3.25, [779] := 3.25, [780] := 3.25,
        [781] := 3.25, [782] := 3.25, [783] := 3.25, [784] := 3.25, [785] := 3.25, [786] := 3.25, [787] := 3.25, [788] := 3.25, [789] := 3.25, [790] := 3.25, [791] := 3.25, [792] := 3.25, [793] := 3.25, [794] := 3.25, [795] := 3.25, [796] := 3.25, [797] := 3.25, [798] := 3.25, [799] := 3.25, [800] := 3.25, [801] := 3.25, [802] := 3.25, [803] := 3.25, [804] := 3.25, [805] := 3.25, [806] := 3.25, [807] := 3.25, [808] := 3.25, [809] := 3.25, [810] := 3.25, [811] := 3.25, [812] := 3.25, [813] := 3.25, [814] := 3.25, [815] := 3.25, [816] := 3.25, [817] := 3.25, [818] := 3.25, [819] := 3.25, [820] := 3.25, [821] := 3.25, [822] := 3.25, [823] := 3.25, [824] := 3.25, [825] := 3.25, [826] := 3.25, [827] := 3.25, [828] := 3.25, [829] := 3.25, [830] := 3.25, [831] := 3.25, [832] := 3.25, [833] := 3.25, [834] := 3.25, [835] := 3.25, [836] := 3.25, [837] := 3.25, [838] := 3.25, [839] := 3.25, [840] := 3.25,
        [841] := 3.25, [842] := 3.25, [843] := 3.25, [844] := 3.25, [845] := 3.25, [846] := 3.25, [847] := 3.25, [848] := 3.25, [849] := 3.25, [850] := 3.25, [851] := 3.25, [852] := 3.25, [853] := 3.25, [854] := 3.25, [855] := 3.25, [856] := 3.25, [857] := 3.25, [858] := 3.25, [859] := 3.25, [860] := 3.25, [861] := 3.25, [862] := 3.25, [863] := 3.25, [864] := 3.25, [865] := 3.25, [866] := 3.25, [867] := 3.25, [868] := 3.25, [869] := 3.25, [870] := 3.25, [871] := 3.25, [872] := 3.25, [873] := 3.25, [874] := 3.25, [875] := 3.25, [876] := 3.25, [877] := 3.25, [878] := 3.25, [879] := 3.25, [880] := 3.25, [881] := 3.25, [882] := 3.25, [883] := 3.25, [884] := 3.25, [885] := 3.25, [886] := 3.25, [887] := 3.25, [888] := 3.25, [889] := 3.25, [890] := 3.25, [891] := 3.25, [892] := 3.25, [893] := 3.25, [894] := 3.25, [895] := 3.25, [896] := 3.25, [897] := 3.25, [898] := 3.25, [899] := 3.25, [900] := 3.25,
        [901] := 3.25, [902] := 3.25, [903] := 3.25, [904] := 3.25, [905] := 3.25, [906] := 3.25, [907] := 3.25, [908] := 3.25, [909] := 3.25, [910] := 3.25, [911] := 3.25, [912] := 3.25, [913] := 3.25, [914] := 3.25, [915] := 3.25, [916] := 3.25, [917] := 3.25, [918] := 3.25, [919] := 3.25, [920] := 3.25, [921] := 3.25, [922] := 3.25, [923] := 3.25, [924] := 3.25, [925] := 3.25, [926] := 3.25, [927] := 3.25, [928] := 3.25, [929] := 3.25, [930] := 3.25, [931] := 3.25, [932] := 3.25, [933] := 3.25, [934] := 3.25, [935] := 3.25, [936] := 3.25, [937] := 3.25, [938] := 3.25, [939] := 3.25, [940] := 3.25, [941] := 3.25, [942] := 3.25, [943] := 3.25, [944] := 3.25, [945] := 3.25, [946] := 3.25, [947] := 3.25, [948] := 3.25, [949] := 3.25, [950] := 3.25, [951] := 3.25, [952] := 3.25, [953] := 3.25, [954] := 3.25, [955] := 3.25, [956] := 3.25, [957] := 3.25, [958] := 3.25, [959] := 3.25, [960] := 3.25,
        [961] := 3.25, [962] := 3.25, [963] := 3.25, [964] := 3.25, [965] := 3.25, [966] := 3.25, [967] := 3.25, [968] := 3.25, [969] := 3.25, [970] := 3.25, [971] := 3.25, [972] := 3.25, [973] := 3.25, [974] := 3.25, [975] := 3.25, [976] := 3.25, [977] := 3.25, [978] := 3.25, [979] := 3.25, [980] := 3.25, [981] := 3.25, [982] := 3.25, [983] := 3.25, [984] := 3.25, [985] := 3.25, [986] := 3.25, [987] := 3.25, [988] := 3.25, [989] := 3.25, [990] := 3.25, [991] := 3.25, [992] := 3.25, [993] := 3.25, [994] := 3.25, [995] := 3.25, [996] := 3.25, [997] := 3.25, [998] := 3.25, [999] := 3.25);
   p29r18_winder_b_selected_diam_inch : REAL := 3.25;   // Winder Winder B Diameter Calculation Selected Diameter [in]
   p29r18_winder_b_unload : REAL := 6.4387383;
   p29r20 : routine := (comment := -1073738505, state := 3);   // Winder Winder Turret VFD
        .FAULT.0   // Winder Liner Winder VFD Drive Fault
        .FAULT.2   // Winder Winder Turret VFD Drive Not Ready
        .FAULT.3   // Winder Winder Turret VFD Drive Not in Remote Mode
        .FAULT.4   // Winder Winder Turret VFD Motor Temperature Fault
        .WARNING.0   // Winder Winder Turret VFD Drive Warning
        .WARNING.1   // Winder Winder Turret VFD No Winder Selected
        .UNACK_FAULT   // Winder Winder Turret VFD Unacknowleged Faults Exist
        .UNACK_WARNING   // Winder Winder Turret VFD Unacknowleged Warnings Exist
        .STATE.0   // Winder Winder Turret One Step Per Scan
        .STATE.1   // Winder Winder Turret Step 1: Idle
        .STATE.2   // Winder Turret Step 2: Start Index Direction
        .STATE.3   // Winder Winder Turret Step 3: Index Active
        .STATE.4   // Winder Winder Turret Step 4: Prox Positive Transition
        .STATE.5   // Winder Winder Turret Step 5: Drive Stop
        .STATE.6   // Winder Winder Turret Step 6: Index Complete
        .STATE.7   // Winder Winder Turret Step 7:Stop Drive
        .STATE.8   // Winder Winder Turret Step 8: Index Complete
   p29r20_acc_dec_ramp : SYS_ACC_DEC_RAMP := (IN_param_master_accel_rate := 2.0, IN_param_master_decel_rate := 2.0, IN_last_scan_s := 0.03426);   // Winder Winder Turret VFD Accel / Decel Ramp
   p29r20_accel_rate : REAL := 2.0;   // Winder Winder Turret VFD Accel Rate
   p29r20_decel_rate : REAL := 2.0;   // Winder Winder Turret VFD Decel Rate
   p29r20_fast_accel : REAL := 2.0;
   p29r20_fast_decel : REAL := 2.0;
   p29r20_index_complete : BOOL := 1;   // Winder Winder Turret VFD Index Complete
   p29r20_index_move_timer : TIMER;   // Winder Winder Turret VFD Move Timer
   p29r20_permissive : BOOL := 1;   // Winder Winder Turret VFD Permissive
   p29r20_request_fwd : BOOL;   // Winder Winder Turret VFD Request Index FWD
   p29r20_request_rev : BOOL;   // Winder Winder Turret VFD Request Index REV
   p29r20_selected_speed : REAL;   // Winder Winder Turret VFD Selected Speed
   p29r20_timer_fault : TIMER[10];   // Winder Winder Turret VFD Fault Dwell Timer
   p29r20_timer_warning : TIMER[4];   // Winder Winder Turret VFD Warning Dwell Timer
   p29r20_zero_speed : BOOL := 1;   // Winder Winder Turret Zero Speed
   p30_di_pin_1 : BOOL := 1;   // Retraction System Inputs Pin 1 Stowed
   p30_di_pin_2 : BOOL := 1;   // Retraction System Inputs Pin 2 Stowed
   p30_di_pin_3 : BOOL := 1;   // Retraction System Inputs Pin 3 Stowed
   p30_di_pin_4 : BOOL := 1;   // Retraction System Inputs Pin 4 Stowed
   p30_di_pin_5 : BOOL := 1;   // Retraction System Inputs Pin 5 Stowed
   p30_di_pin_6 : BOOL := 1;   // Retraction System Inputs Pin 6 Stowed
   p30_di_pin_7 : BOOL := 1;   // Retraction System Inputs Pin 7 Stowed
   p30_di_pin_8 : BOOL := 1;   // Retraction System Inputs Pin 8 Stowed
   p30_di_retraction_down_ls : BOOL;   // Retraction System Digital Input LS: Down
   p30_di_retraction_up_ls : BOOL;   // Retraction System Digital Input Operator Side LS: Up
   p30_di_rotation_fault : BOOL;   // Retraction System Digital Input Rotation Fault
   p30_di_ss_close : BOOL;   // Retraction System Digital Input SS: Open/Off/Close Close
   p30_di_ss_open : BOOL;   // Retraction System Digital Input SS: Open/Off/Close Open
   p30_dint_to_hmi : DINT[16] := ([0] := 255);   // Retraction System Dint to HMI
        [0].0   // Retraction System Dint to HMI Safety Pin 1 Stowed
        [0].1   // Retraction System Dint to HMI Safety Pin 2 Stowed
        [0].2   // Retraction System Dint to HMI Safety Pin 3 Stowed
        [0].3   // Retraction System Dint to HMI Safety Pin 4 Stowed
        [0].4   // Retraction System Dint to HMI Safety Pin 5 Stowed
        [0].5   // Retraction System Dint to HMI Safety Pin 6 Stowed
        [0].6   // Retraction System Dint to HMI Safety Pin 7 Stowed
        [0].7   // Retraction System Dint to HMI Safety Pin 8 Stowed
        [2].0   // Retraction System Alarms A00: Rotation Fault
        [2].1   // Retraction System Alarms A01:
        [2].2   // Retraction System Alarms A02:
        [2].3   // Retraction System Alarms A03:
        [2].4   // Retraction System Alarms A04:
        [2].5   // Retraction System Alarms A05:
        [2].6   // Retraction System Alarms A06:
        [2].7   // Retraction System Alarms A07:
        [2].8   // Retraction System Alarms A08:
        [2].9   // Retraction System Alarms A09
        [2].10   // Retraction System Alarms A10:
        [2].11   // Retraction System Alarms A11:
        [2].12   // Retraction System Alarms A12:
        [2].13   // Retraction System Alarms A13:
        [2].14   // Retraction System Alarms A14:
        [2].15   // Retraction System Alarms A15:
        [2].16   // Retraction System Alarms A16:
        [2].17   // Retraction System Alarms A17:
        [2].18   // Retraction System Alarms A18:
        [2].19   // Retraction System Alarms A19:
        [2].20   // Retraction System Alarms A20:
        [2].21   // Retraction System Alarms A21:
        [2].22   // Retraction System Alarms A22:
        [2].23   // Retraction System Alarms A23:
        [2].24   // Retraction System Alarms A24:
        [2].25   // Retraction System Alarms A25:
        [2].26   // Retraction System Alarms A26:
        [2].27   // Retraction System Alarms A27:
        [2].28   // Retraction System Alarms A28:
        [2].29   // Retraction System Alarms A29:
        [2].30   // Retraction System Alarms A30:
        [2].31   // Retraction System Alarms A31:
        [4].0   // Retraction System Warnings W00:
        [4].1   // Retraction System Warnings W01:
        [4].2   // Retraction System Warnings W02:
        [4].3   // Retraction System Warnings W03:
        [4].4   // Retraction System Warnings W04:
        [4].5   // Retraction System Warnings W05:
        [4].6   // Retraction System Warnings W06:
        [4].7   // Retraction System Warnings W07:
        [4].8   // Retraction System Warnings W08:
        [4].9   // Retraction System Warnings W09
        [4].10   // Retraction System Warnings W10:
        [4].11   // Retraction System Warnings W11:
        [4].12   // Retraction System Warnings W12:
        [4].13   // Retraction System Warnings W13:
        [4].14   // Retraction System Warnings W14:
        [4].15   // Retraction System Warnings W15:
        [4].16   // Retraction System Warnings W16:
        [4].17   // Retraction System Warnings W17:
        [4].18   // Retraction System Warnings W18:
        [4].19   // Retraction System Warnings W19:
        [4].20   // Retraction System Warnings W20:
        [4].21   // Retraction System Warnings W21:
        [4].22   // Retraction System Warnings W22:
        [4].23   // Retraction System Warnings W23:
        [4].24   // Retraction System Warnings W24:
        [4].25   // Retraction System Warnings W25:
        [4].26   // Retraction System Warnings W26:
        [4].27   // Retraction System Warnings W27:
        [4].28   // Retraction System Warnings W28:
        [4].29   // Retraction System Warnings W29:
        [4].30   // Retraction System Warnings W30:
        [4].31   // Retraction System Warnings W31:
   p30_do_retract_motion : BOOL;
   p30_do_retract_reset : BOOL;
   p30_do_rotation_fwd : BOOL;   // Retraction System Output Retraction FWD
   p30_do_rotation_rev : BOOL;   // Retraction System Output Retraction REV
   p30_real_to_hmi : REAL[112];   // Retraction System Real to HMI
   p30r01 : routine := (comment := 7);   // Retraction System
   p30r02 : routine := (comment := -1073741761);   // Retraction System Misc Control
   p30r02_fault_exists : BOOL;
   p30r02_timer_fault : TIMER[4];   // Retraction System Misc Control Fault Dwell Timer
   p30r02_timer_warning : TIMER[4];   // Retraction System Misc Control Warning Dwell Timer
   p30r02_unack_fault : BOOL;   // Retraction System Misc Control Unacknoledged Fault Exist
   p30r02_unack_warning : BOOL;   // Retraction System Misc Control Unacknoledge Warning Exist
   p30r02_warning_exists : BOOL;
   p30r03 : routine := (comment := -1073741761);   // Retraction System Input
   p30r03_timer_fault : TIMER[4];   // Retraction System Input Fault Dwell Timer
   p30r03_timer_warning : TIMER[4];   // Retraction System Input Warning Dwell Timer
   p30r04 : routine := (comment := -1073741761);   // Retraction System Output
   p30r04_timer_fault : TIMER[4];   // Retraction System Output Fault Dwell Timer
   p30r04_timer_warning : TIMER[4];   // Retraction System Output Warning Dwell Timer
   p30r05 : routine := (comment := -1073741761);   // Retraction System Dint to HMI
   p30r05_timer_fault : TIMER[4];   // Retraction System Dint to HMI Fault Dwell Timer
   p30r05_timer_warning : TIMER[4];   // Retraction System Dint to HMI Warning Dwell Timer
   p30r06 : routine := (comment := -1073741572);   // Retraction System Real to HMI
   p30r06_timer_fault : TIMER[4];   // Retraction System Real to HMI Fault Dwell Timer
   p30r06_timer_warning : TIMER[4];   // Retraction System Real to HMI Warning Dwell Timer
   p30r07 : routine := (comment := -1073741761);   // Retraction System Alarms
   p30r07_timer_fault : TIMER[4];   // Retraction System Alarms Fault Dwell Timer
   p30r07_timer_warning : TIMER[4];   // Retraction System Alarms Warning Dwell Timer
   p30r08 : routine := (comment := -1073741761);   // Retraction System Warnings
   p30r08_timer_fault : TIMER[4];   // Retraction System Warnings Fault Dwell Timer
   p30r08_timer_warning : TIMER[4];   // Retraction System Warnings Warning Dwell Timer
   p30r09 : routine := (comment := -1073741761);   // Retraction System Modes
   p30r09_mode_close : BOOL;   // Retraction System Modes Close Mode
   p30r09_mode_off : BOOL := 1;   // Retraction System Modes Off Mode
   p30r09_mode_open : BOOL;   // Retraction System Modes Open Mode
   p30r09_timer_fault : TIMER[4];   // Retraction System Modes Fault Dwell Timer
   p30r09_timer_warning : TIMER[4];   // Retraction System Modes Warning Dwell Timer
   p30r10 : routine := (comment := -1073741777);   // Retraction System Retraction
        .FAULT.0   // Retraction System Retraction Rotation Fault
        .WARNING.0   // Retraction System Retraction Pins Not Stowed
   p30r10_motion_monitor_dwell : TIMER := (PRE := 500);
   p30r10_request_close : BOOL;   // Retraction System Retraction Request Close
   p30r10_request_monitor : BOOL;
   p30r10_request_open : BOOL;   // Retraction System Retraction Request Open
   p30r10_run_permissive : BOOL := 1;   // Retraction System Retraction Run Permissive
   p30r10_safety_pins_stowed : BOOL := 1;   // Retraction System Retraction All Safety Pins Stowed
   p30r10_state : DINT;   // Splice Press Sequence State
        .0   // Splice Press Sequence State 0 One Step Per Scan
        .1   // Splice Press Sequence State 1 Idle
        .2   // Splice Press Sequence State 2 Enable Sequence
        .3   // Splice Press Sequence State 3 Close Exit Clamp
        .4   // Splice Press Sequence State 4 Close Inlet Clamp
        .5   // Splice Press Sequence State 5 Closing Platen
        .6   // Splice Press Sequence State 6 Cure in Progress
        .7   // Splice Press Sequence State 7 Cure Done
        .8   // Splice Press Sequence State 8 Platen Open
        .9   // Splice Press Sequence State 9 Inlet Clamp Open
        .10   // Splice Press Sequence State 10 Exit Clamp Open
        .11   // Splice Press Sequence State 11 Complete
   p30r10_timer_fault : TIMER[4] := ([1].PRE := 400);   // Retraction System Retraction Fault Dwell Timer
   p30r10_timer_warning : TIMER[4] := ([0].PRE := 1000);   // Retraction System Retraction Warning Dwell Timer
   p31r09 : routine;   // Edge Control Modes
        .UNACK_FAULT   // Edge Control Modes Unacknowledged Fault Exists
        .UNACK_WARNING   // Edge Control Modes Unacknowledged Warning Exists
   p32r13_request_auto_stop : BOOL;   // Impreg Supply VFD Request Auto Stop
   retraction_delay_timer : TIMER := (PRE := 4000);
   retraction_delay_timer_2 : TIMER := (PRE := 4000);
   spring_spd_adj_prcnt : REAL := 0.975;
   turret_in_position : BOOL := 1;   // Turret In Position
   winder_ramped_setpoint : REAL;
END_VAR

PROGRAM P01_Main   (* main routine R01_Main *)
VAR
   PIDE_02 : PID_ENHANCED := (PV := 60.0, PVEUMax := 500.0, SPProg := 102.227806, SPOper := 102.227806, SPHLimit := 200.0, RatioProg := 1.0, RatioOper := 1.0, RatioHLimit := 1.0, RatioLLimit := 1.0, CVProg := 50.0, CVOper := 100.0, CVEUMax := 100.0, CVHLimit := 100.0, PGain := 5.0, IGain := 0.1, PVEDerivative := 1, DSmoothing := 1, PVTracking := 1, PVHHLimit := 1000.0, PVHLimit := 900.0, PVLLimit := -1000.0, PVLLLimit := -2000.0, DevHHLimit := 1000.0, DevHLimit := 1000.0, ManualAfterInit := 1, ProgAutoReq := 1, RTSTime := 1, CVEU := 100.0, CV := 100.0, CVHAlarm := 1, SP := 102.227806, SPPercent := 20.44556, PVPercent := 12.0, E := 42.227806, EPercent := 8.44556, InitPrimary := 1, WindupHOut := 1, Ratio := 1.0, DevLAlarm := 1, DevLLAlarm := 1, ProgOper := 1, Auto := 1, DeltaT := 0.1, AtuneBusy := 1);
END_VAR

ROUTINE R01_Main   (* ladder *)
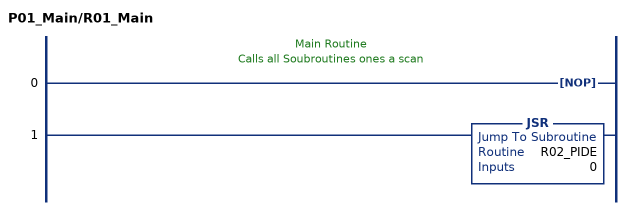
   // Main Routine
   // Calls all Soubroutines ones a scan
   0: NOP();
   1: JSR(R02_PIDE,0);
END_ROUTINE

ROUTINE R02_PIDE   (* function block diagram *)
   SHEET 1
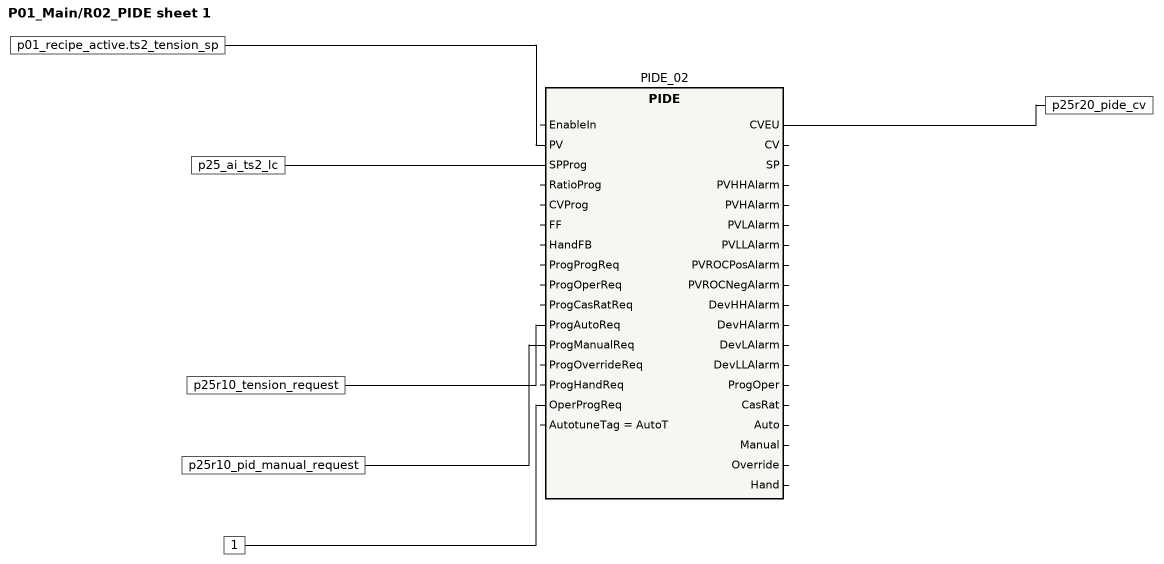
   PIDE_02 : PIDE(PV := p01_recipe_active.ts2_tension_sp, SPProg := p25_ai_ts2_lc, ProgAutoReq := p25r10_tension_request, ProgManualReq := p25r10_pid_manual_request, OperProgReq := 1, AutotuneTag := AutoT);   // unwired pins: EnableIn RatioProg CVProg FF HandFB ProgProgReq ProgOperReq ProgCasRatReq ProgOverrideReq ProgHandReq CV SP PVHHAlarm PVHAlarm PVLAlarm PVLLAlarm PVROCPosAlarm PVROCNegAlarm DevHHAlarm DevHAlarm DevLAlarm DevLLAlarm ProgOper CasRat Auto Manual Override Hand
   p25r20_pide_cv := PIDE_02.CVEU;
END_ROUTINE
END_PROGRAM

PROGRAM P01_System   (* main routine R01_Main *)
VAR
   Limit_Clamp : sys_Limit_Clamp;   // Limit Clamp
   tmrFlash : TIMER[4] := ([0].PRE := 1000, [0].ACC := 365, [0].EN := 1, [0].TT := 1, [1].PRE := 1000, [2].PRE := 500, [2].ACC := 530, [2].EN := 1, [2].DN := 1, [3].PRE := 500, [3].ACC := 500, [3].EN := 1, [3].DN := 1);   // Flash Timer
END_VAR

ROUTINE R01_Main   (* ladder *)
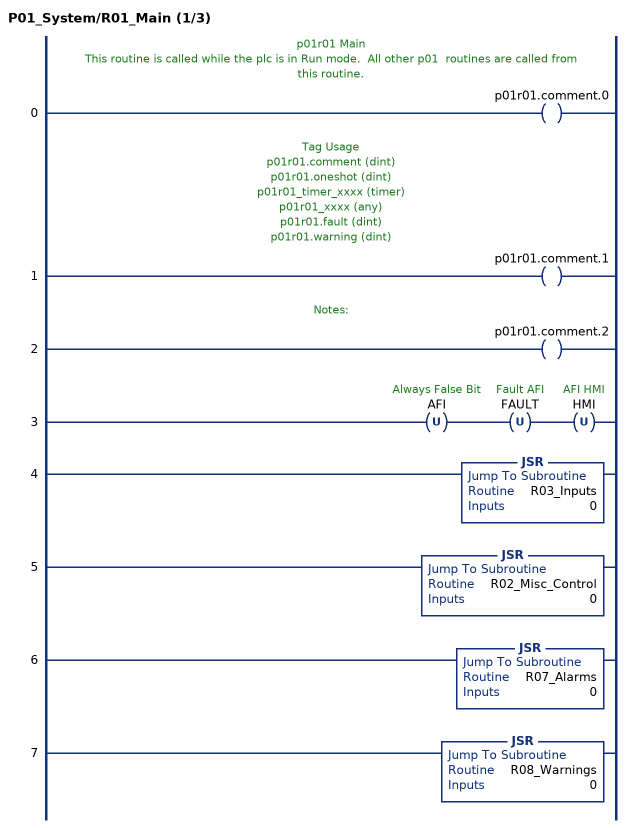
   // p01r01 Main
   // This routine is called while the plc is in Run mode.  All other p01  routines are called from this routine.
   0: OTE(p01r01.comment.0);
   // Tag Usage
   // p01r01.comment (dint)
   // p01r01.oneshot (dint)
   // p01r01_timer_xxxx (timer)
   // p01r01_xxxx (any)
   // p01r01.fault (dint)
   // p01r01.warning (dint)
   1: OTE(p01r01.comment.1);
   // Notes:
   2: OTE(p01r01.comment.2);
   3: OTU(AFI)OTU(FAULT)OTU(HMI);
   4: JSR(R03_Inputs,0);
   5: JSR(R02_Misc_Control,0);
   6: JSR(R07_Alarms,0);
   7: JSR(R08_Warnings,0);
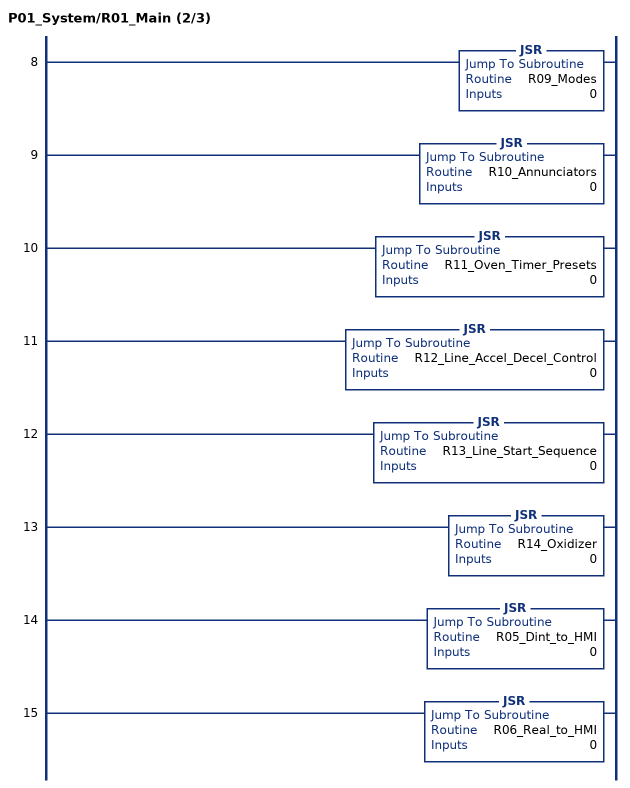
   8: JSR(R09_Modes,0);
   9: JSR(R10_Annunciators,0);
   10: JSR(R11_Oven_Timer_Presets,0);
   11: JSR(R12_Line_Accel_Decel_Control,0);
   12: JSR(R13_Line_Start_Sequence,0);
   13: JSR(R14_Oxidizer,0);
   14: JSR(R05_Dint_to_HMI,0);
   15: JSR(R06_Real_to_HMI,0);
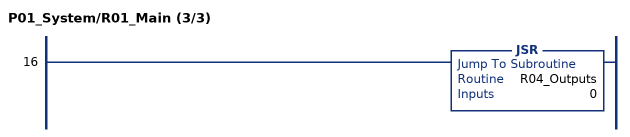
   16: JSR(R04_Outputs,0);
END_ROUTINE

ROUTINE R02_Misc_Control   (* ladder *)
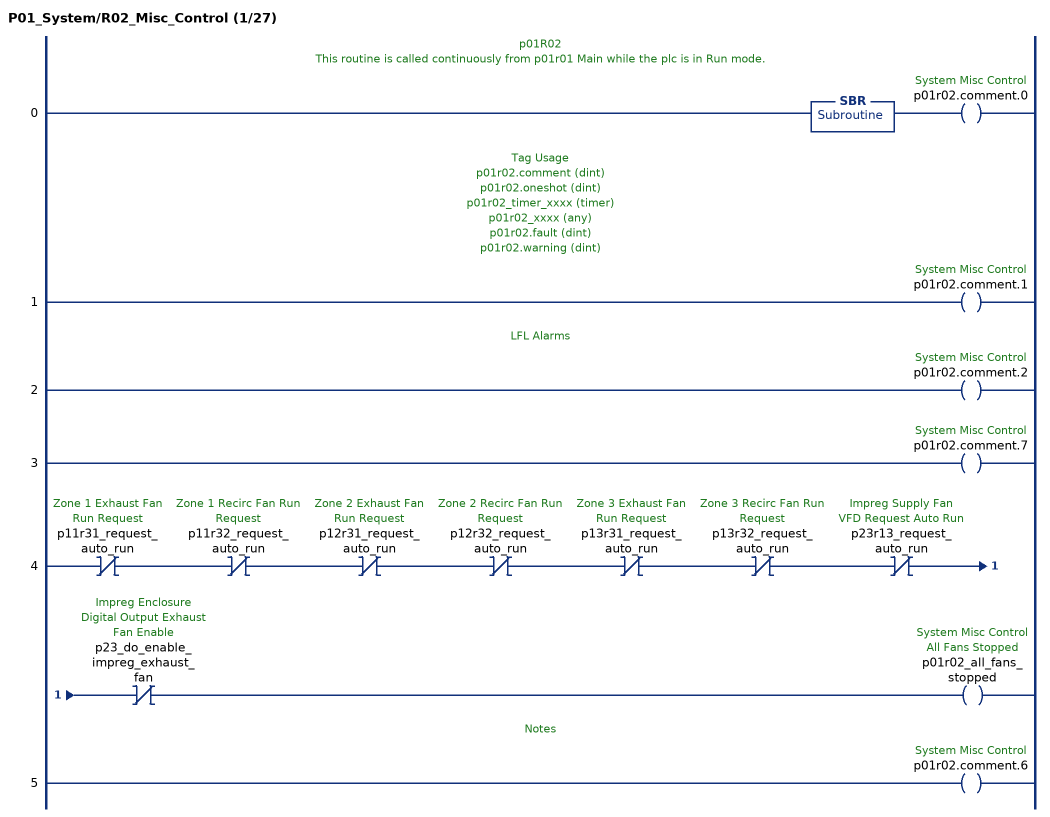
   // p01R02
   // This routine is called continuously from p01r01 Main while the plc is in Run mode.
   0: SBR()OTE(p01r02.comment.0);
   // Tag Usage
   // p01r02.comment (dint)
   // p01r02.oneshot (dint)
   // p01r02_timer_xxxx (timer)
   // p01r02_xxxx (any)
   // p01r02.fault (dint)
   // p01r02.warning (dint)
   1: OTE(p01r02.comment.1);
   // LFL Alarms
   2: OTE(p01r02.comment.2);
   3: OTE(p01r02.comment.7);
   4: XIO(p11r31_request_auto_run)XIO(p11r32_request_auto_run)XIO(p12r31_request_auto_run)XIO(p12r32_request_auto_run)XIO(p13r31_request_auto_run)XIO(p13r32_request_auto_run)XIO(p23r13_request_auto_run)XIO(p23_do_enable_impreg_exhaust_fan)OTE(p01r02_all_fans_stopped);
   // Notes
   5: OTE(p01r02.comment.6);
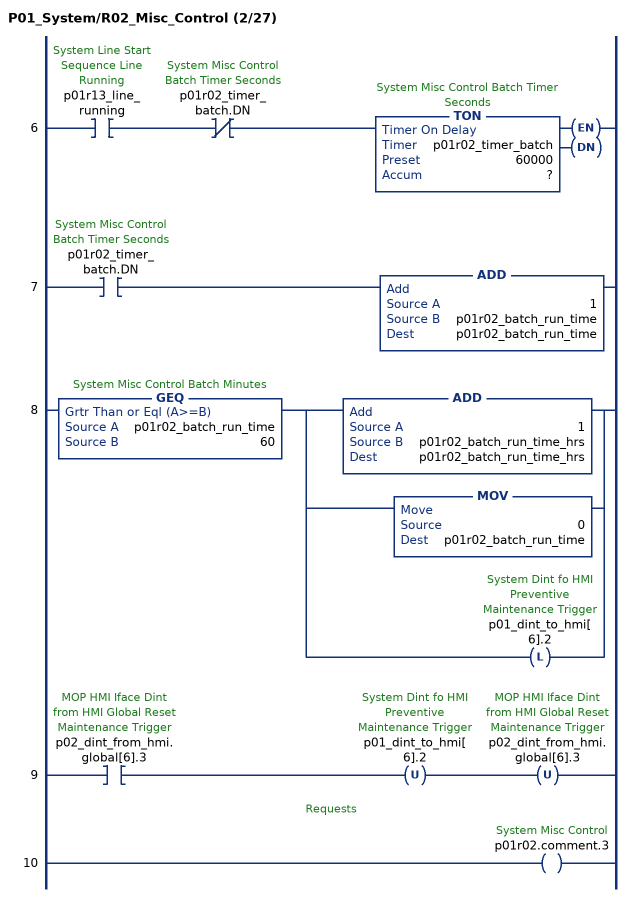
   6: XIC(p01r13_line_running)XIO(p01r02_timer_batch.DN)TON(p01r02_timer_batch,?,?);
   7: XIC(p01r02_timer_batch.DN)ADD(1,p01r02_batch_run_time,p01r02_batch_run_time);
   8: GEQ(p01r02_batch_run_time,60)[ADD(1,p01r02_batch_run_time_hrs,p01r02_batch_run_time_hrs) ,MOV(0,p01r02_batch_run_time) ,OTL(p01_dint_to_hmi[6].2) ];
   9: XIC(p02_dint_from_hmi.global[6].3)OTU(p01_dint_to_hmi[6].2)OTU(p02_dint_from_hmi.global[6].3);
   // Requests
   10: OTE(p01r02.comment.3);
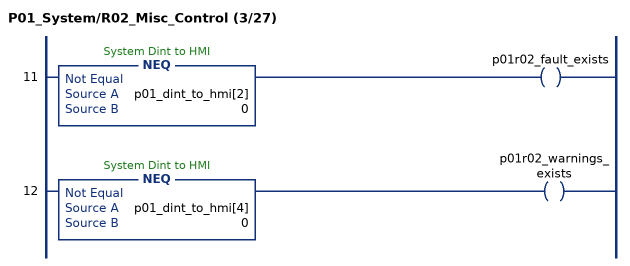
   11: NEQ(p01_dint_to_hmi[2],0)OTE(p01r02_fault_exists);
   12: NEQ(p01_dint_to_hmi[4],0)OTE(p01r02_warnings_exists);
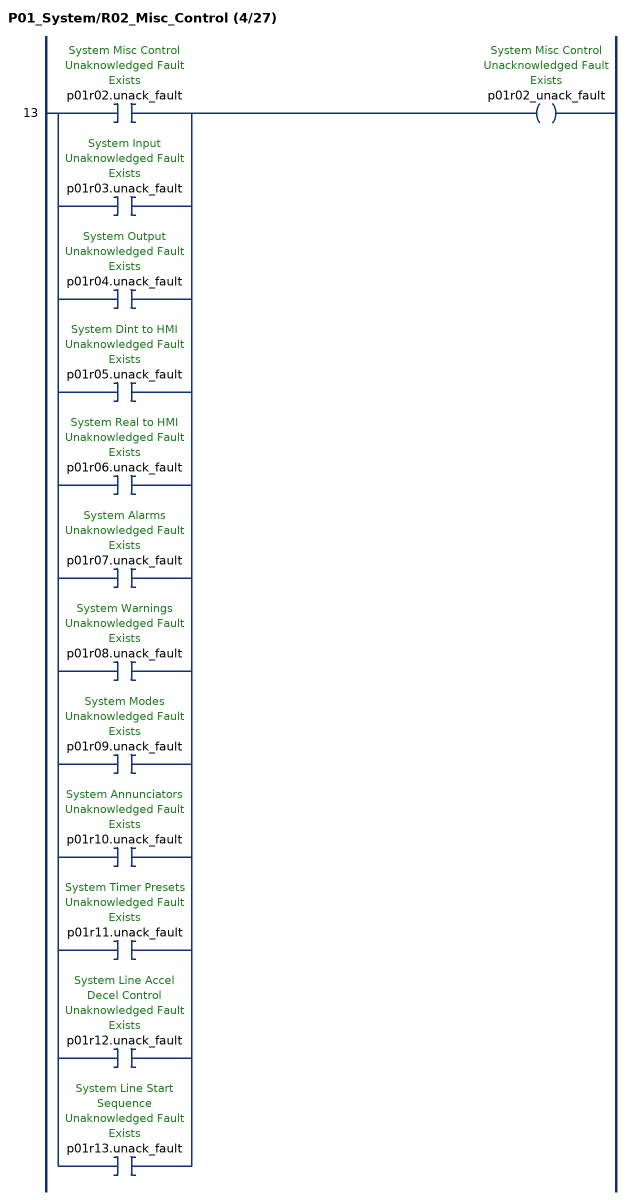
   13: [XIC(p01r02.unack_fault) ,XIC(p01r03.unack_fault) ,XIC(p01r04.unack_fault) ,XIC(p01r05.unack_fault) ,XIC(p01r06.unack_fault) ,XIC(p01r07.unack_fault) ,XIC(p01r08.unack_fault) ,XIC(p01r09.unack_fault) ,XIC(p01r10.unack_fault) ,XIC(p01r11.unack_fault) ,XIC(p01r12.unack_fault) ,XIC(p01r13.unack_fault) ]OTE(p01r02_unack_fault);
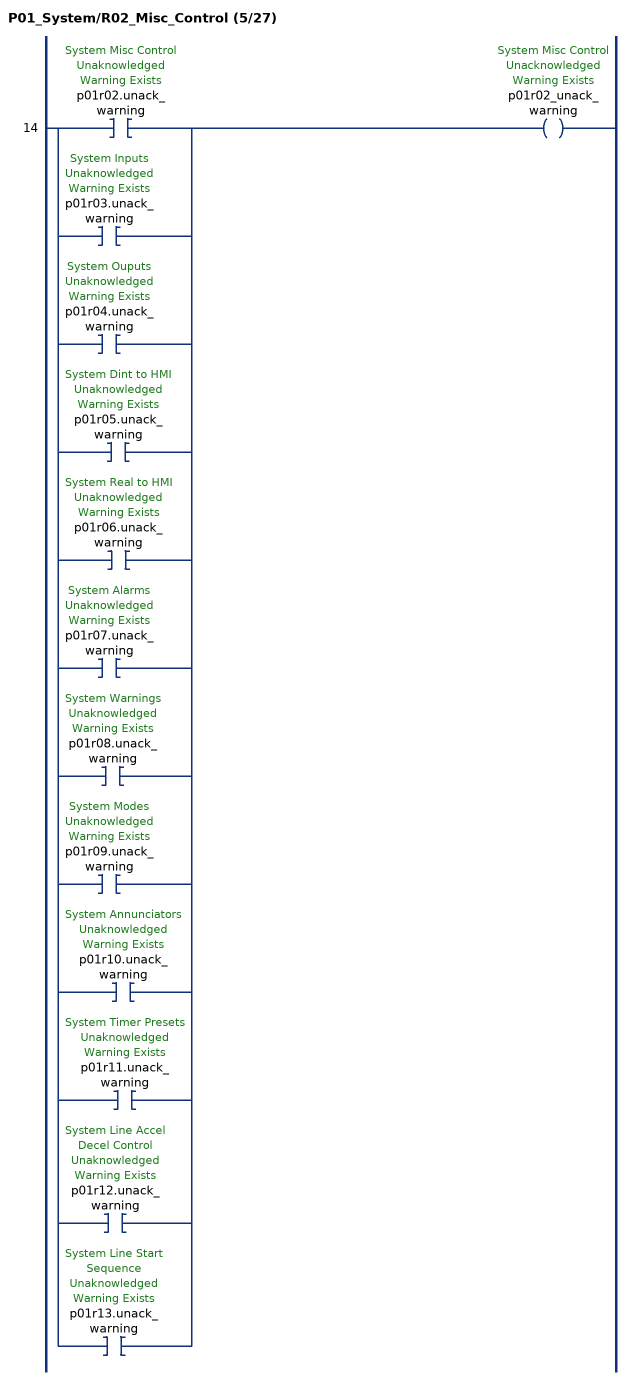
   14: [XIC(p01r02.unack_warning) ,XIC(p01r03.unack_warning) ,XIC(p01r04.unack_warning) ,XIC(p01r05.unack_warning) ,XIC(p01r06.unack_warning) ,XIC(p01r07.unack_warning) ,XIC(p01r08.unack_warning) ,XIC(p01r09.unack_warning) ,XIC(p01r10.unack_warning) ,XIC(p01r11.unack_warning) ,XIC(p01r12.unack_warning) ,XIC(p01r13.unack_warning) ]OTE(p01r02_unack_warning);
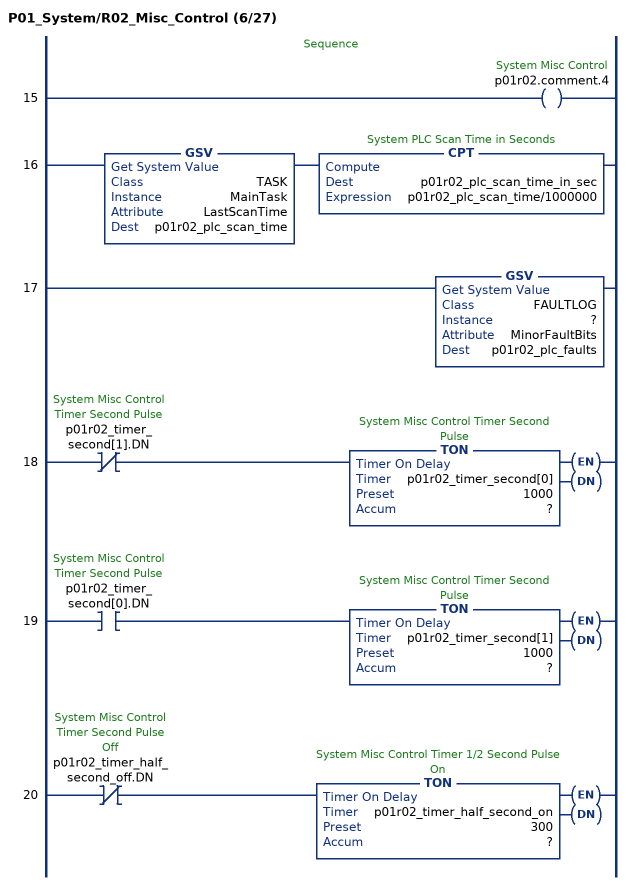
   // Sequence
   15: OTE(p01r02.comment.4);
   16: GSV(TASK,MainTask,LastScanTime,p01r02_plc_scan_time)CPT(p01r02_plc_scan_time_in_sec,p01r02_plc_scan_time/1000000);
   17: GSV(FAULTLOG,?,MinorFaultBits,p01r02_plc_faults);
   18: XIO(p01r02_timer_second[1].DN)TON(p01r02_timer_second[0],?,?);
   19: XIC(p01r02_timer_second[0].DN)TON(p01r02_timer_second[1],?,?);
   20: XIO(p01r02_timer_half_second_off.DN)TON(p01r02_timer_half_second_on,?,?);
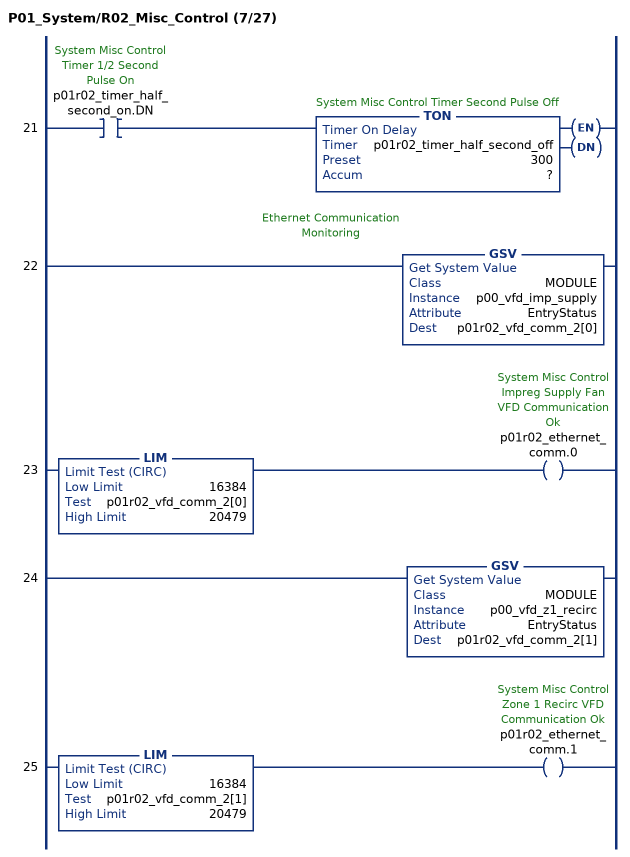
   21: XIC(p01r02_timer_half_second_on.DN)TON(p01r02_timer_half_second_off,?,?);
   // Ethernet Communication
   // Monitoring
   22: GSV(MODULE,p00_vfd_imp_supply,EntryStatus,p01r02_vfd_comm_2[0]);
   23: LIM(16384,p01r02_vfd_comm_2[0],20479)OTE(p01r02_ethernet_comm.0);
   24: GSV(MODULE,p00_vfd_z1_recirc,EntryStatus,p01r02_vfd_comm_2[1]);
   25: LIM(16384,p01r02_vfd_comm_2[1],20479)OTE(p01r02_ethernet_comm.1);
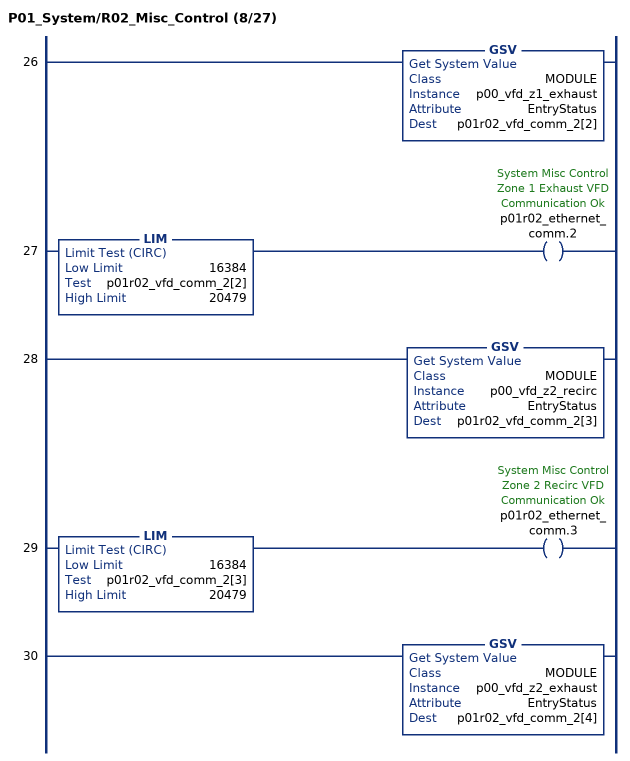
   26: GSV(MODULE,p00_vfd_z1_exhaust,EntryStatus,p01r02_vfd_comm_2[2]);
   27: LIM(16384,p01r02_vfd_comm_2[2],20479)OTE(p01r02_ethernet_comm.2);
   28: GSV(MODULE,p00_vfd_z2_recirc,EntryStatus,p01r02_vfd_comm_2[3]);
   29: LIM(16384,p01r02_vfd_comm_2[3],20479)OTE(p01r02_ethernet_comm.3);
   30: GSV(MODULE,p00_vfd_z2_exhaust,EntryStatus,p01r02_vfd_comm_2[4]);
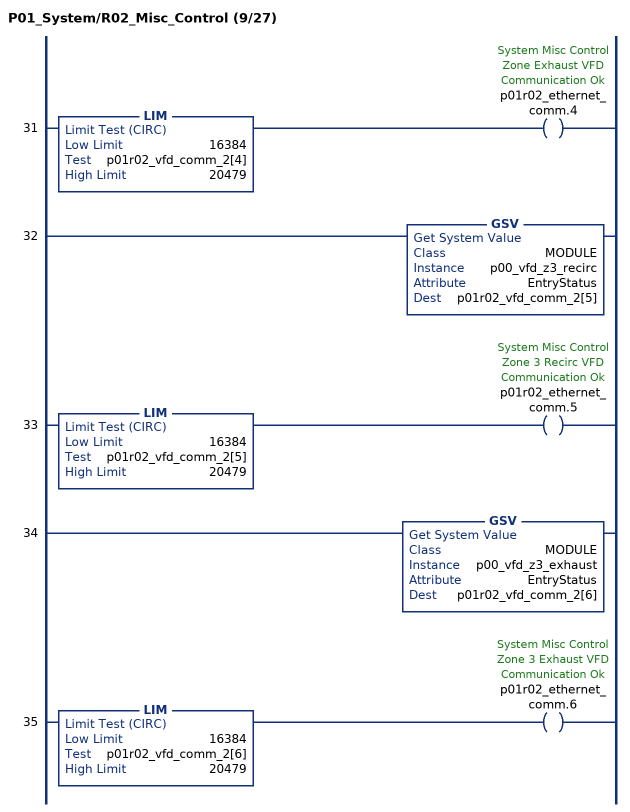
   31: LIM(16384,p01r02_vfd_comm_2[4],20479)OTE(p01r02_ethernet_comm.4);
   32: GSV(MODULE,p00_vfd_z3_recirc,EntryStatus,p01r02_vfd_comm_2[5]);
   33: LIM(16384,p01r02_vfd_comm_2[5],20479)OTE(p01r02_ethernet_comm.5);
   34: GSV(MODULE,p00_vfd_z3_exhaust,EntryStatus,p01r02_vfd_comm_2[6]);
   35: LIM(16384,p01r02_vfd_comm_2[6],20479)OTE(p01r02_ethernet_comm.6);
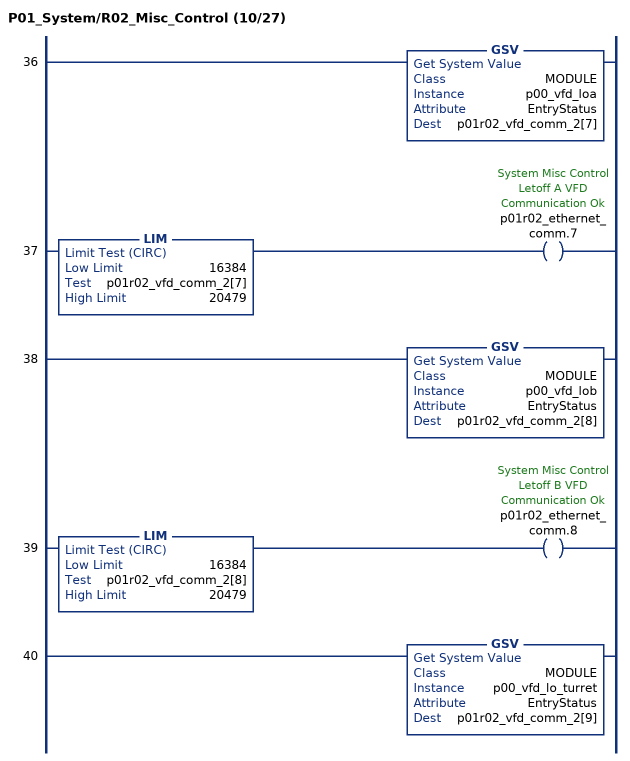
   36: GSV(MODULE,p00_vfd_loa,EntryStatus,p01r02_vfd_comm_2[7]);
   37: LIM(16384,p01r02_vfd_comm_2[7],20479)OTE(p01r02_ethernet_comm.7);
   38: GSV(MODULE,p00_vfd_lob,EntryStatus,p01r02_vfd_comm_2[8]);
   39: LIM(16384,p01r02_vfd_comm_2[8],20479)OTE(p01r02_ethernet_comm.8);
   40: GSV(MODULE,p00_vfd_lo_turret,EntryStatus,p01r02_vfd_comm_2[9]);
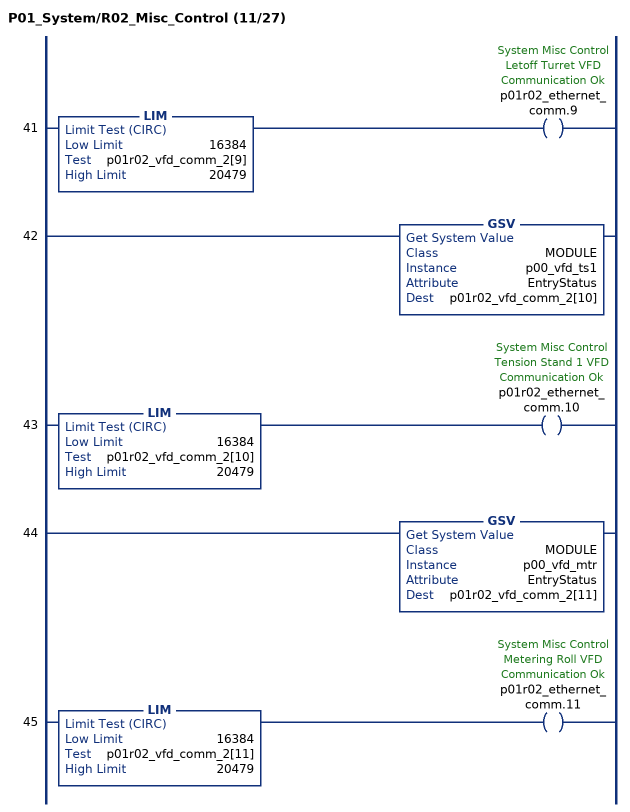
   41: LIM(16384,p01r02_vfd_comm_2[9],20479)OTE(p01r02_ethernet_comm.9);
   42: GSV(MODULE,p00_vfd_ts1,EntryStatus,p01r02_vfd_comm_2[10]);
   43: LIM(16384,p01r02_vfd_comm_2[10],20479)OTE(p01r02_ethernet_comm.10);
   44: GSV(MODULE,p00_vfd_mtr,EntryStatus,p01r02_vfd_comm_2[11]);
   45: LIM(16384,p01r02_vfd_comm_2[11],20479)OTE(p01r02_ethernet_comm.11);
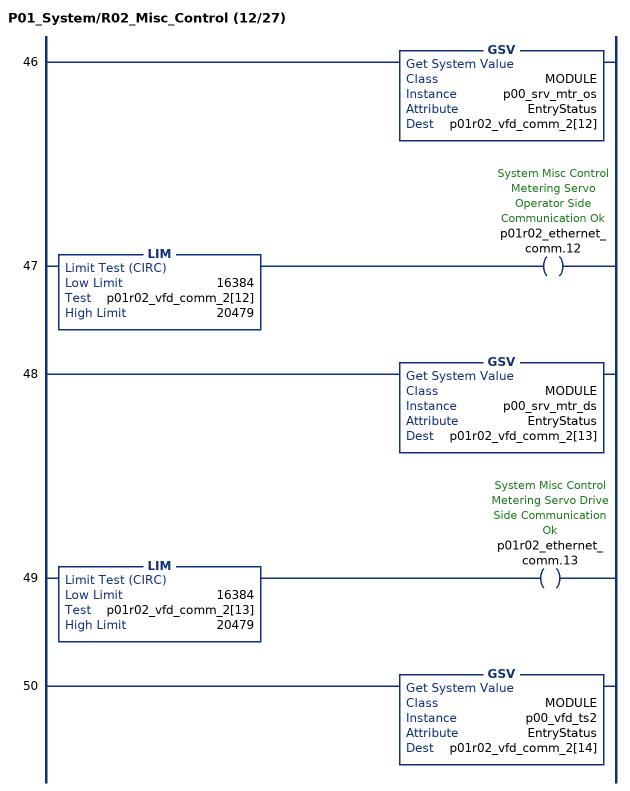
   46: GSV(MODULE,p00_srv_mtr_os,EntryStatus,p01r02_vfd_comm_2[12]);
   47: LIM(16384,p01r02_vfd_comm_2[12],20479)OTE(p01r02_ethernet_comm.12);
   48: GSV(MODULE,p00_srv_mtr_ds,EntryStatus,p01r02_vfd_comm_2[13]);
   49: LIM(16384,p01r02_vfd_comm_2[13],20479)OTE(p01r02_ethernet_comm.13);
   50: GSV(MODULE,p00_vfd_ts2,EntryStatus,p01r02_vfd_comm_2[14]);
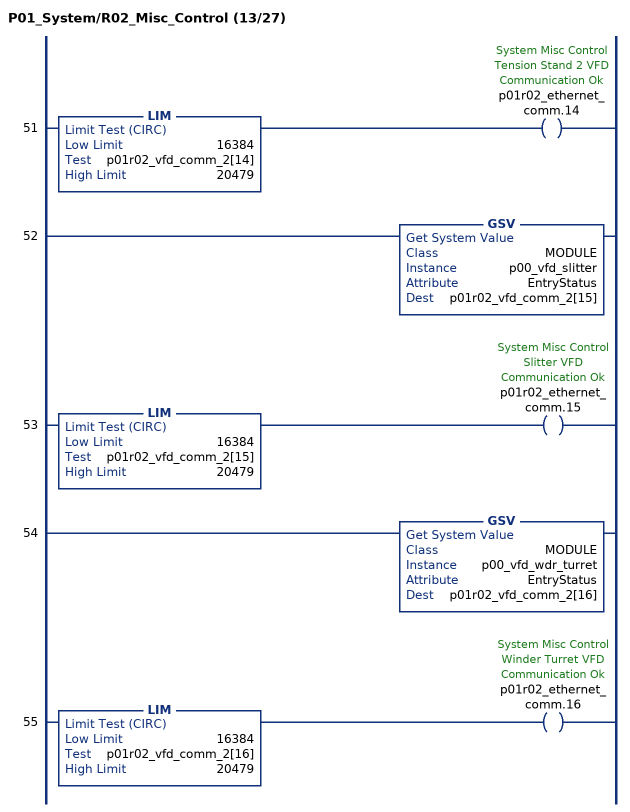
   51: LIM(16384,p01r02_vfd_comm_2[14],20479)OTE(p01r02_ethernet_comm.14);
   52: GSV(MODULE,p00_vfd_slitter,EntryStatus,p01r02_vfd_comm_2[15]);
   53: LIM(16384,p01r02_vfd_comm_2[15],20479)OTE(p01r02_ethernet_comm.15);
   54: GSV(MODULE,p00_vfd_wdr_turret,EntryStatus,p01r02_vfd_comm_2[16]);
   55: LIM(16384,p01r02_vfd_comm_2[16],20479)OTE(p01r02_ethernet_comm.16);
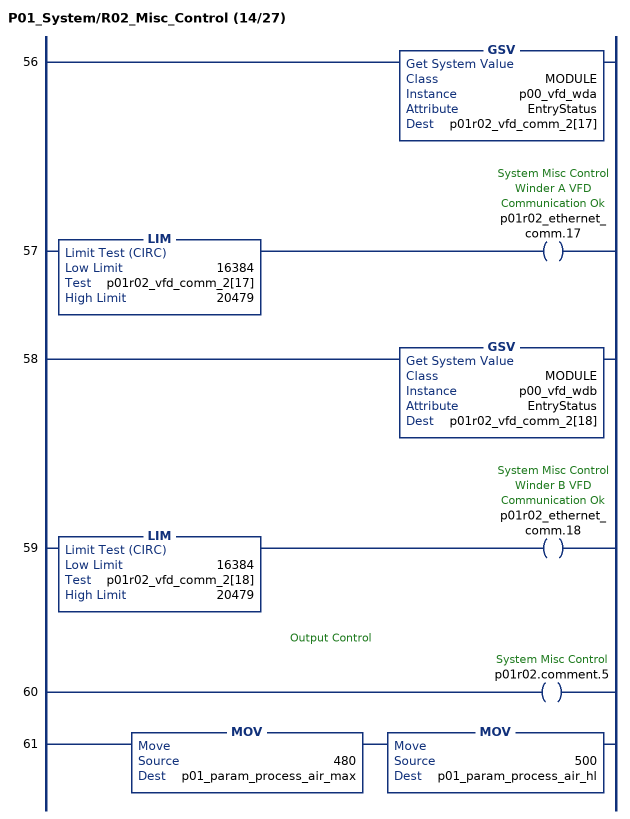
   56: GSV(MODULE,p00_vfd_wda,EntryStatus,p01r02_vfd_comm_2[17]);
   57: LIM(16384,p01r02_vfd_comm_2[17],20479)OTE(p01r02_ethernet_comm.17);
   58: GSV(MODULE,p00_vfd_wdb,EntryStatus,p01r02_vfd_comm_2[18]);
   59: LIM(16384,p01r02_vfd_comm_2[18],20479)OTE(p01r02_ethernet_comm.18);
   // Output Control
   60: OTE(p01r02.comment.5);
   61: MOV(480,p01_param_process_air_max)MOV(500,p01_param_process_air_hl);
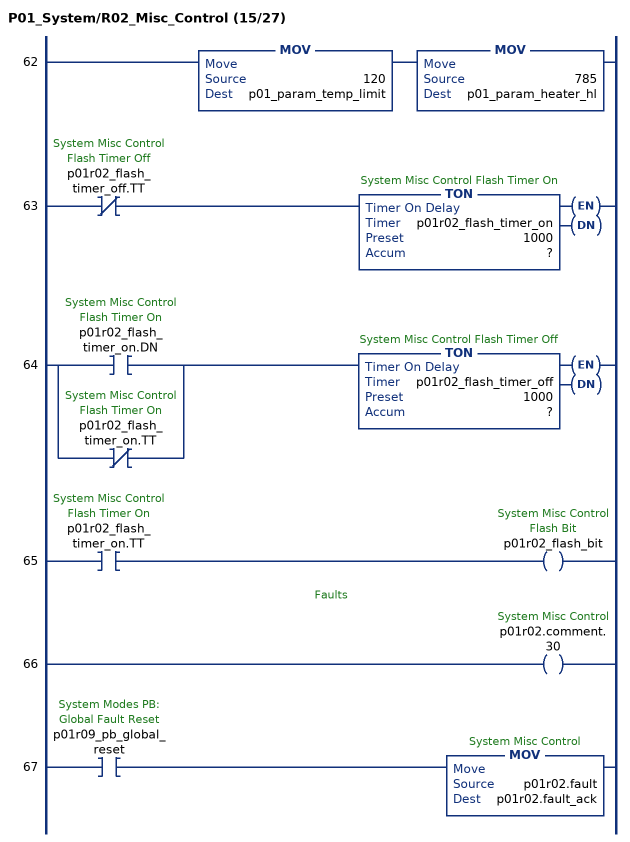
   62: MOV(120,p01_param_temp_limit)MOV(785,p01_param_heater_hl);
   63: XIO(p01r02_flash_timer_off.TT)TON(p01r02_flash_timer_on,?,?);
   64: [XIC(p01r02_flash_timer_on.DN) ,XIO(p01r02_flash_timer_on.TT) ]TON(p01r02_flash_timer_off,?,?);
   65: XIC(p01r02_flash_timer_on.TT)OTE(p01r02_flash_bit);
   // Faults
   66: OTE(p01r02.comment.30);
   67: XIC(p01r09_pb_global_reset)MOV(p01r02.fault,p01r02.fault_ack);
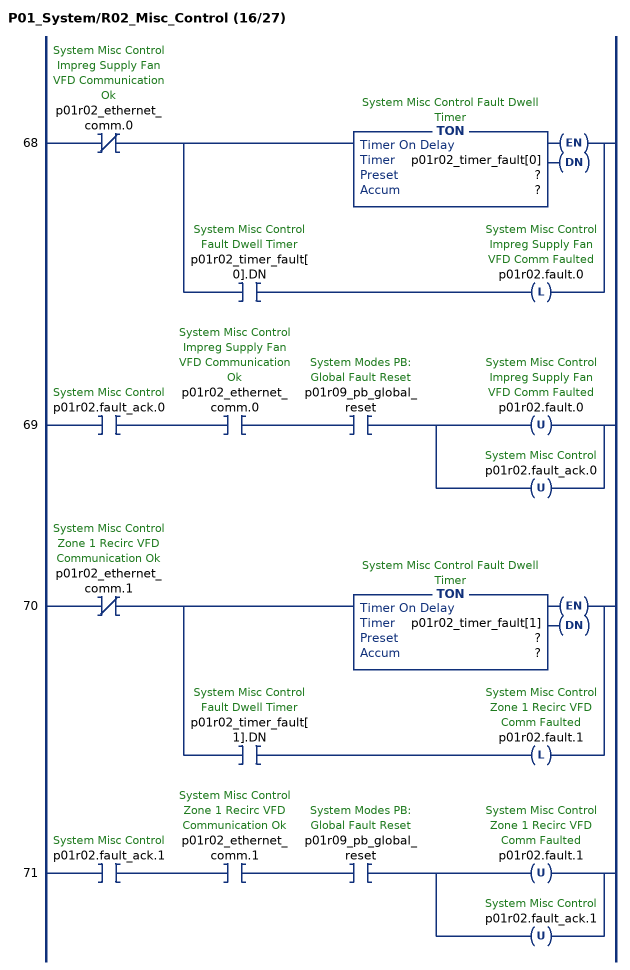
   68: XIO(p01r02_ethernet_comm.0)[TON(p01r02_timer_fault[0],?,?) ,XIC(p01r02_timer_fault[0].DN) OTL(p01r02.fault.0) ];
   69: XIC(p01r02.fault_ack.0)XIC(p01r02_ethernet_comm.0)XIC(p01r09_pb_global_reset)[OTU(p01r02.fault.0) ,OTU(p01r02.fault_ack.0) ];
   70: XIO(p01r02_ethernet_comm.1)[TON(p01r02_timer_fault[1],?,?) ,XIC(p01r02_timer_fault[1].DN) OTL(p01r02.fault.1) ];
   71: XIC(p01r02.fault_ack.1)XIC(p01r02_ethernet_comm.1)XIC(p01r09_pb_global_reset)[OTU(p01r02.fault.1) ,OTU(p01r02.fault_ack.1) ];
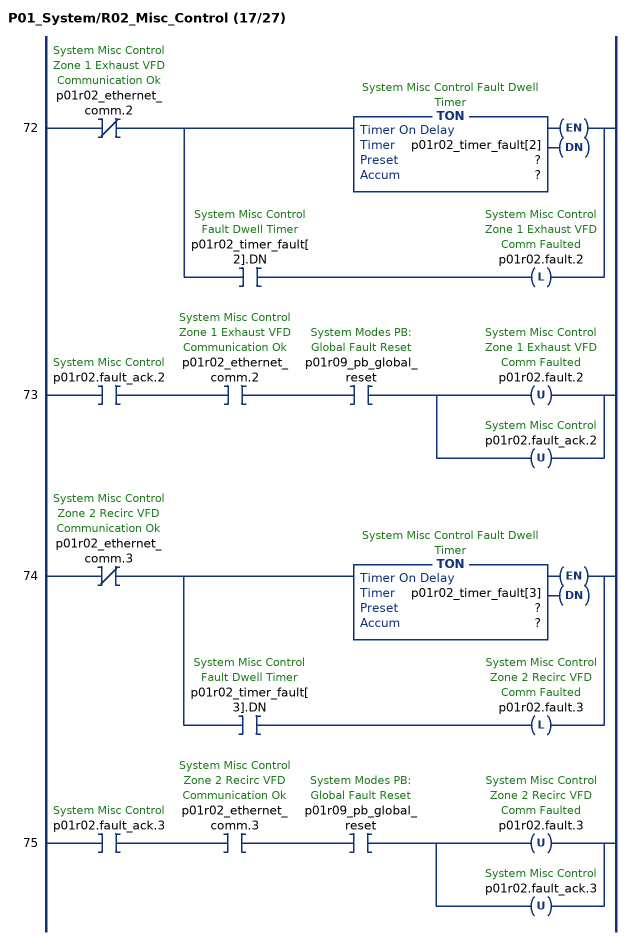
   72: XIO(p01r02_ethernet_comm.2)[TON(p01r02_timer_fault[2],?,?) ,XIC(p01r02_timer_fault[2].DN) OTL(p01r02.fault.2) ];
   73: XIC(p01r02.fault_ack.2)XIC(p01r02_ethernet_comm.2)XIC(p01r09_pb_global_reset)[OTU(p01r02.fault.2) ,OTU(p01r02.fault_ack.2) ];
   74: XIO(p01r02_ethernet_comm.3)[TON(p01r02_timer_fault[3],?,?) ,XIC(p01r02_timer_fault[3].DN) OTL(p01r02.fault.3) ];
   75: XIC(p01r02.fault_ack.3)XIC(p01r02_ethernet_comm.3)XIC(p01r09_pb_global_reset)[OTU(p01r02.fault.3) ,OTU(p01r02.fault_ack.3) ];
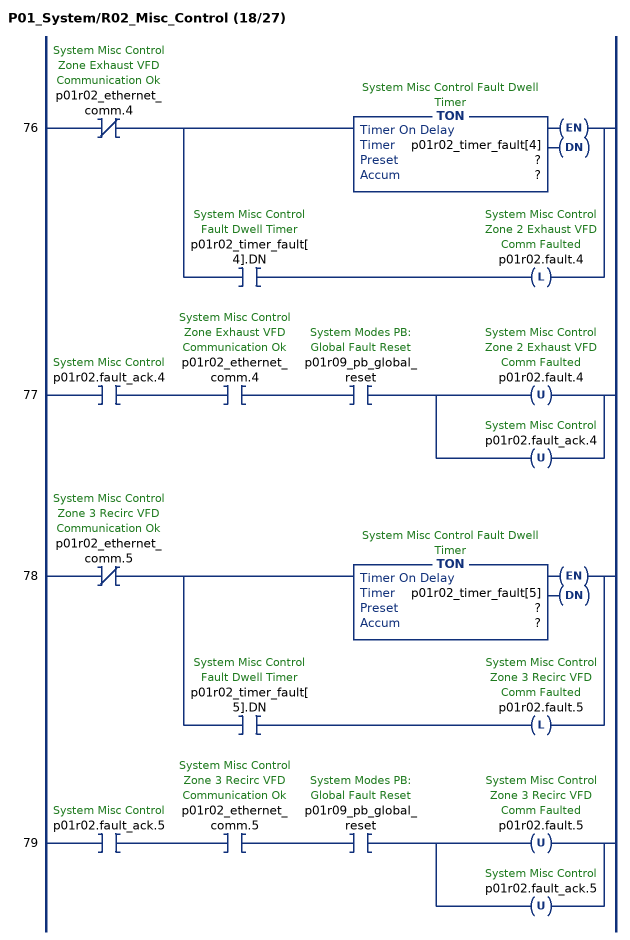
   76: XIO(p01r02_ethernet_comm.4)[TON(p01r02_timer_fault[4],?,?) ,XIC(p01r02_timer_fault[4].DN) OTL(p01r02.fault.4) ];
   77: XIC(p01r02.fault_ack.4)XIC(p01r02_ethernet_comm.4)XIC(p01r09_pb_global_reset)[OTU(p01r02.fault.4) ,OTU(p01r02.fault_ack.4) ];
   78: XIO(p01r02_ethernet_comm.5)[TON(p01r02_timer_fault[5],?,?) ,XIC(p01r02_timer_fault[5].DN) OTL(p01r02.fault.5) ];
   79: XIC(p01r02.fault_ack.5)XIC(p01r02_ethernet_comm.5)XIC(p01r09_pb_global_reset)[OTU(p01r02.fault.5) ,OTU(p01r02.fault_ack.5) ];
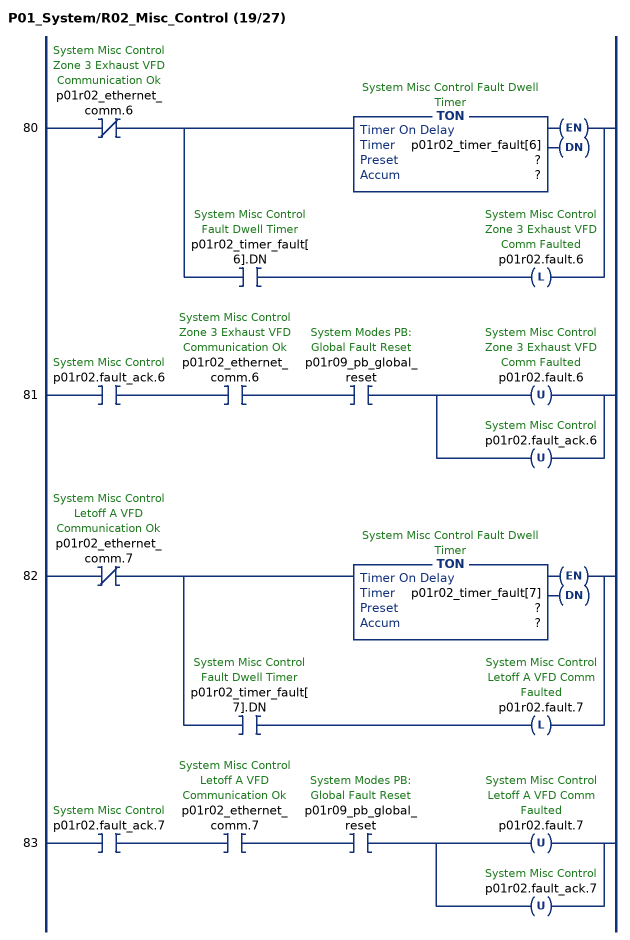
   80: XIO(p01r02_ethernet_comm.6)[TON(p01r02_timer_fault[6],?,?) ,XIC(p01r02_timer_fault[6].DN) OTL(p01r02.fault.6) ];
   81: XIC(p01r02.fault_ack.6)XIC(p01r02_ethernet_comm.6)XIC(p01r09_pb_global_reset)[OTU(p01r02.fault.6) ,OTU(p01r02.fault_ack.6) ];
   82: XIO(p01r02_ethernet_comm.7)[TON(p01r02_timer_fault[7],?,?) ,XIC(p01r02_timer_fault[7].DN) OTL(p01r02.fault.7) ];
   83: XIC(p01r02.fault_ack.7)XIC(p01r02_ethernet_comm.7)XIC(p01r09_pb_global_reset)[OTU(p01r02.fault.7) ,OTU(p01r02.fault_ack.7) ];
